LIN {X 0,Y 298.54,Z 403.296,A -85,B 0,C 180,E1 -16483.61,E2 -16483.61} C_VEL
LIN {X 0,Y 298.534,Z 403.297,A -85,B 0,C 180,E1 -16486.404,E2 -16486.404} C_VEL
LIN {X 0,Y 298.495,Z 403.302,A -85,B 0,C 180,E1 -16489.65,E2 -16489.65} C_VEL
LIN {X 0,Y 298.401,Z 403.314,A -85,B 0,C 180,E1 -16493.596,E2 -16493.596} C_VEL
LIN {X 0,Y 298.321,Z 403.323,A -85,B 0,C 180,E1 -16496.584,E2 -16496.584} C_VEL
LIN {X 0,Y 297.954,Z 403.371,A -85,B 0,C 180,E1 -16499.685,E2 -16499.685} C_VEL
LIN {X 0,Y 297.517,Z 403.428,A -85,B 0,C 180,E1 -16502.902,E2 -16502.902} C_VEL
LIN {X 0,Y 297.315,Z 403.659,A -85,B 0,C 180,E1 -16504.556,E2 -16504.556} C_VEL
LIN {X 0,Y 297.205,Z 406.502,A -85,B 0,C 180,E1 -16507.931,E2 -16507.931} C_VEL
LIN {X 0,Y 297.211,Z 408.026,A -85,B 0,C 180,E1 -16509.558,E2 -16509.558} C_VEL
LIN {X 0,Y 300.389,Z 421.173,A -85,B 0,C 180,E1 -16510.429,E2 -16510.429} C_VEL
LIN {X 0,Y 303.208,Z 434.297,A -85,B 0,C 180,E1 -16511.559,E2 -16511.559} C_VEL
LIN {X 0,Y 304.476,Z 441.111,A -85,B 0,C 180,E1 -16512.256,E2 -16512.256} C_VEL
LIN {X 0,Y 303.235,Z 453.565,A -85,B 0,C 180,E1 -16513.594,E2 -16513.594} C_VEL
LIN {X 0,Y 302.004,Z 464.15,A -85,B 0,C 180,E1 -16515.022,E2 -16515.022} C_VEL
LIN {X 0,Y 300.91,Z 473.555,A -85,B 0,C 180,E1 -16516.59,E2 -16516.59} C_VEL
LIN {X 0,Y 299.618,Z 483.514,A -85,B 0,C 180,E1 -16518.634,E2 -16518.634} C_VEL
LIN {X 0,Y 298.679,Z 491.025,A -85,B 0,C 180,E1 -16520.558,E2 -16520.558} C_VEL
LIN {X 0,Y 297.874,Z 498.058,A -85,B 0,C 180,E1 -16522.831,E2 -16522.831} C_VEL
LIN {X 0,Y 297.405,Z 502.476,A -85,B 0,C 180,E1 -16524.624,E2 -16524.624} C_VEL
LIN {X 0,Y 296.973,Z 507.02,A -85,B 0,C 180,E1 -16527.024,E2 -16527.024} C_VEL
LIN {X 0,Y 296.702,Z 509.213,A -85,B 0,C 180,E1 -16528.594,E2 -16528.594} C_VEL
LIN {X 0,Y 296.597,Z 511.611,A -85,B 0,C 180,E1 -16531.237,E2 -16531.237} C_VEL
LIN {X 0,Y 296.595,Z 512.398,A -85,B 0,C 180,E1 -16533.244,E2 -16533.244} C_VEL
LIN {X 0,Y 296.774,Z 512.436,A -85,B 0,C 180,E1 -16534.771,E2 -16534.771} C_VEL
LIN {X 0,Y 297.237,Z 511.374,A -85,B 0,C 180,E1 -16537.223,E2 -16537.223} C_VEL
LIN {X 0,Y 297.865,Z 509.479,A -85,B 0,C 180,E1 -16539.274,E2 -16539.274} C_VEL
LIN {X 0,Y 298.691,Z 506.354,A -85,B 0,C 180,E1 -16541.481,E2 -16541.481} C_VEL
LIN {X 0,Y 299.914,Z 501.581,A -85,B 0,C 180,E1 -16543.874,E2 -16543.874} C_VEL
LIN {X 0,Y 301.541,Z 495.408,A -85,B 0,C 180,E1 -16546.18,E2 -16546.18} C_VEL
LIN {X 0,Y 303.291,Z 488.055,A -85,B 0,C 180,E1 -16548.303,E2 -16548.303} C_VEL
LIN {X 0,Y 305.109,Z 480.486,A -85,B 0,C 180,E1 -16550.053,E2 -16550.053} C_VEL
LIN {X 0,Y 307.147,Z 471.173,A -85,B 0,C 180,E1 -16551.823,E2 -16551.823} C_VEL
LIN {X 0,Y 309.342,Z 460.153,A -85,B 0,C 180,E1 -16553.479,E2 -16553.479} C_VEL
LIN {X 0,Y 310.412,Z 454.213,A -85,B 0,C 180,E1 -16554.23,E2 -16554.23} C_VEL
LIN {X 0,Y 310.495,Z 451.09,A -85,B 0,C 180,E1 -16554.656,E2 -16554.656} C_VEL
LIN {X 0,Y 309.213,Z 446.849,A -85,B 0,C 180,E1 -16555.373,E2 -16555.373} C_VEL
LIN {X 0,Y 306.912,Z 443.084,A -85,B 0,C 180,E1 -16556.121,E2 -16556.121} C_VEL
LIN {X 0,Y 301.408,Z 435.464,A -85,B 0,C 180,E1 -16557.657,E2 -16557.657} C_VEL
LIN {X 0,Y 299.994,Z 432.52,A -85,B 0,C 180,E1 -16558.139,E2 -16558.139} C_VEL
LIN {X 0,Y 294.566,Z 419.508,A -85,B 0,C 180,E1 -16560.087,E2 -16560.087} C_VEL
LIN {X 0,Y 293.298,Z 416.848,A -85,B 0,C 180,E1 -16560.473,E2 -16560.473} C_VEL
LIN {X 0,Y 292.122,Z 413.899,A -85,B 0,C 180,E1 -16560.863,E2 -16560.863} C_VEL
LIN {X 0,Y 292.037,Z 413.448,A -85,B 0,C 180,E1 -16560.949,E2 -16560.949} C_VEL
LIN {X 0,Y 292.102,Z 411.884,A -85,B 0,C 180,E1 -16564.14,E2 -16564.14} C_VEL
LIN {X 0,Y 292.37,Z 410.624,A -85,B 0,C 180,E1 -16566.904,E2 -16566.904} C_VEL
LIN {X 0,Y 292.432,Z 409.493,A -85,B 0,C 180,E1 -16569.859,E2 -16569.859} C_VEL
LIN {X 0,Y 292.138,Z 408.34,A -85,B 0,C 180,E1 -16573.921,E2 -16573.921} C_VEL
LIN {X 0,Y 292.041,Z 407.747,A -85,B 0,C 180,E1 -16576.786,E2 -16576.786} C_VEL
LIN {X 0,Y 291.975,Z 407.316,A -85,B 0,C 180,E1 -16580.177,E2 -16580.177} C_VEL
LIN {X 0,Y 291.967,Z 407.269,A -85,B 0,C 180,E1 -16584.156,E2 -16584.156} C_VEL
LIN {X 0,Y 292.013,Z 407.587,A -85,B 0,C 180,E1 -16587.213,E2 -16587.213} C_VEL
LIN {X 0,Y 292.068,Z 408.231,A -85,B 0,C 180,E1 -16590.354,E2 -16590.354} C_VEL
LIN {X 0,Y 292.244,Z 409.294,A -85,B 0,C 180,E1 -16593.582,E2 -16593.582} C_VEL
LIN {X 0,Y 292.592,Z 411.114,A -85,B 0,C 180,E1 -16597.577,E2 -16597.577} C_VEL
LIN {X 0,Y 292.906,Z 412.784,A -85,B 0,C 180,E1 -16600.38,E2 -16600.38} C_VEL
LIN {X 0,Y 293.404,Z 415.441,A -85,B 0,C 180,E1 -16604.07,E2 -16604.07} C_VEL
LIN {X 0,Y 293.953,Z 418.857,A -85,B 0,C 180,E1 -16607.985,E2 -16607.985} C_VEL
LIN {X 0,Y 294.409,Z 422.603,A -85,B 0,C 180,E1 -16611.644,E2 -16611.644} C_VEL
LIN {X 0,Y 294.307,Z 425.693,A -85,B 0,C 180,E1 -16614.285,E2 -16614.285} C_VEL
LIN {X 0,Y 293.028,Z 430.824,A -85,B 0,C 180,E1 -16618.16,E2 -16618.16} C_VEL
LIN {X 0,Y 292.222,Z 434.847,A -85,B 0,C 180,E1 -16621.038,E2 -16621.038} C_VEL
LIN {X 0,Y 293.241,Z 438.506,A -85,B 0,C 180,E1 -16621.432,E2 -16621.432} C_VEL
LIN {X 0,Y 296.189,Z 447.824,A -85,B 0,C 180,E1 -16622.521,E2 -16622.521} C_VEL
LIN {X 0,Y 299.074,Z 460.374,A -85,B 0,C 180,E1 -16623.974,E2 -16623.974} C_VEL
LIN {X 0,Y 300.545,Z 472.286,A -85,B 0,C 180,E1 -16625.426,E2 -16625.426} C_VEL
LIN {X 0,Y 300.842,Z 482.738,A -85,B 0,C 180,E1 -16626.789,E2 -16626.789} C_VEL
LIN {X 0,Y 300.143,Z 492.535,A -85,B 0,C 180,E1 -16628.184,E2 -16628.184} C_VEL
LIN {X 0,Y 298.035,Z 501.95,A -85,B 0,C 180,E1 -16629.652,E2 -16629.652} C_VEL
LIN {X 0,Y 295.564,Z 512.297,A -85,B 0,C 180,E1 -16631.641,E2 -16631.641} C_VEL
LIN {X 0,Y 293.71,Z 520.668,A -85,B 0,C 180,E1 -16633.676,E2 -16633.676} C_VEL
LIN {X 0,Y 292.256,Z 527.544,A -85,B 0,C 180,E1 -16635.736,E2 -16635.736} C_VEL
LIN {X 0,Y 290.836,Z 533.963,A -85,B 0,C 180,E1 -16638.153,E2 -16638.153} C_VEL
LIN {X 0,Y 290.116,Z 538.211,A -85,B 0,C 180,E1 -16640.242,E2 -16640.242} C_VEL
LIN {X 0,Y 289.828,Z 540.46,A -85,B 0,C 180,E1 -16641.64,E2 -16641.64} C_VEL
LIN {X 0,Y 289.518,Z 543.698,A -85,B 0,C 180,E1 -16644.433,E2 -16644.433} C_VEL
LIN {X 0,Y 289.534,Z 544.718,A -85,B 0,C 180,E1 -16645.829,E2 -16645.829} C_VEL
LIN {X 0,Y 289.561,Z 545.291,A -85,B 0,C 180,E1 -16647.223,E2 -16647.223} C_VEL
LIN {X 0,Y 289.811,Z 545.227,A -85,B 0,C 180,E1 -16650.005,E2 -16650.005} C_VEL
LIN {X 0,Y 289.704,Z 544.575,A -85,B 0,C 180,E1 -16651.395,E2 -16651.395} C_VEL
LIN {X 0,Y 289.616,Z 543.459,A -85,B 0,C 180,E1 -16652.787,E2 -16652.787} C_VEL
LIN {X 0,Y 289.663,Z 541.916,A -85,B 0,C 180,E1 -16654.179,E2 -16654.179} C_VEL
LIN {X 0,Y 289.681,Z 539.425,A -85,B 0,C 180,E1 -16655.888,E2 -16655.888} C_VEL
LIN {X 0,Y 289.868,Z 534.452,A -85,B 0,C 180,E1 -16658.37,E2 -16658.37} C_VEL
LIN {X 0,Y 290.274,Z 528.94,A -85,B 0,C 180,E1 -16660.467,E2 -16660.467} C_VEL
LIN {X 0,Y 290.98,Z 522.039,A -85,B 0,C 180,E1 -16662.56,E2 -16662.56} C_VEL
LIN {X 0,Y 291.798,Z 514.992,A -85,B 0,C 180,E1 -16664.297,E2 -16664.297} C_VEL
LIN {X 0,Y 292.636,Z 506.875,A -85,B 0,C 180,E1 -16665.961,E2 -16665.961} C_VEL
LIN {X 0,Y 294.068,Z 497.254,A -85,B 0,C 180,E1 -16667.566,E2 -16667.566} C_VEL
LIN {X 0,Y 295.416,Z 485.913,A -85,B 0,C 180,E1 -16669.098,E2 -16669.098} C_VEL
LIN {X 0,Y 294.777,Z 474.417,A -85,B 0,C 180,E1 -16670.412,E2 -16670.412} C_VEL
LIN {X 0,Y 293.431,Z 461.228,A -85,B 0,C 180,E1 -16671.612,E2 -16671.612} C_VEL
LIN {X 0,Y 291.781,Z 447.799,A -85,B 0,C 180,E1 -16672.555,E2 -16672.555} C_VEL
LIN {X 0,Y 290.651,Z 439.673,A -85,B 0,C 180,E1 -16673.019,E2 -16673.019} C_VEL
LIN {X 0,Y 291.447,Z 432.932,A -85,B 0,C 180,E1 -16677.274,E2 -16677.274} C_VEL
LIN {X 0,Y 292.325,Z 426.915,A -85,B 0,C 180,E1 -16681.129,E2 -16681.129} C_VEL
LIN {X 0,Y 293.176,Z 422.072,A -85,B 0,C 180,E1 -16684.292,E2 -16684.292} C_VEL
LIN {X 0,Y 293.704,Z 418.403,A -85,B 0,C 180,E1 -16686.748,E2 -16686.748} C_VEL
LIN {X 0,Y 293.176,Z 413.948,A -85,B 0,C 180,E1 -16689.904,E2 -16689.904} C_VEL
LIN {X 0,Y 292.115,Z 408.18,A -85,B 0,C 180,E1 -16694.249,E2 -16694.249} C_VEL
LIN {X 0,Y 291.373,Z 404.192,A -85,B 0,C 180,E1 -16697.516,E2 -16697.516} C_VEL
LIN {X 0,Y 291.351,Z 404.195,A -85,B 0,C 180,E1 -16701.157,E2 -16701.157} C_VEL
LIN {X 0,Y 291.372,Z 404.188,A -85,B 0,C 180,E1 -16704.626,E2 -16704.626} C_VEL
LIN {X 0,Y 291.383,Z 404.186,A -85,B 0,C 180,E1 -16707.951,E2 -16707.951} C_VEL
LIN {X 0,Y 291.362,Z 404.193,A -85,B 0,C 180,E1 -16711.155,E2 -16711.155} C_VEL
LIN {X 0,Y 291.376,Z 404.186,A -85,B 0,C 180,E1 -16714.267,E2 -16714.267} C_VEL
LIN {X 0,Y 291.38,Z 404.19,A -85,B 0,C 180,E1 -16717.298,E2 -16717.298} C_VEL
LIN {X 0,Y 291.408,Z 404.183,A -85,B 0,C 180,E1 -16720.265,E2 -16720.265} C_VEL
LIN {X 0,Y 291.515,Z 404.172,A -85,B 0,C 180,E1 -16724.665,E2 -16724.665} C_VEL
LIN {X 0,Y 291.545,Z 404.17,A -85,B 0,C 180,E1 -16728.88,E2 -16728.88} C_VEL
LIN {X 0,Y 291.682,Z 404.149,A -85,B 0,C 180,E1 -16731.687,E2 -16731.687} C_VEL
LIN {X 0,Y 291.627,Z 404.157,A -85,B 0,C 180,E1 -16734.467,E2 -16734.467} C_VEL
LIN {X 0,Y 291.9,Z 404.124,A -85,B 0,C 180,E1 -16738.619,E2 -16738.619} C_VEL
LIN {X 0,Y 291.896,Z 404.124,A -85,B 0,C 180,E1 -16741.378,E2 -16741.378} C_VEL
LIN {X 0,Y 291.701,Z 404.151,A -85,B 0,C 180,E1 -16746.918,E2 -16746.918} C_VEL
LIN {X 0,Y 291.582,Z 404.161,A -85,B 0,C 180,E1 -16749.712,E2 -16749.712} C_VEL
LIN {X 0,Y 291.528,Z 404.168,A -85,B 0,C 180,E1 -16753.949,E2 -16753.949} C_VEL
LIN {X 0,Y 291.441,Z 404.184,A -85,B 0,C 180,E1 -16756.819,E2 -16756.819} C_VEL
LIN {X 0,Y 291.405,Z 404.184,A -85,B 0,C 180,E1 -16759.84,E2 -16759.84} C_VEL
LIN {X 0,Y 291.394,Z 404.185,A -85,B 0,C 180,E1 -16764.204,E2 -16764.204} C_VEL
LIN {X 0,Y 291.424,Z 404.182,A -85,B 0,C 180,E1 -16767.27,E2 -16767.27} C_VEL
LIN {X 0,Y 291.334,Z 404.195,A -85,B 0,C 180,E1 -16770.436,E2 -16770.436} C_VEL
LIN {X 0,Y 291.354,Z 404.189,A -85,B 0,C 180,E1 -16773.695,E2 -16773.695} C_VEL
LIN {X 0,Y 291.378,Z 404.187,A -85,B 0,C 180,E1 -16777.249,E2 -16777.249} C_VEL
LIN {X 0,Y 291.34,Z 404.196,A -85,B 0,C 180,E1 -16780.639,E2 -16780.639} C_VEL
LIN {X 0,Y 291.299,Z 404.201,A -85,B 0,C 180,E1 -16784.398,E2 -16784.398} C_VEL
LIN {X 0,Y 291.324,Z 404.197,A -85,B 0,C 180,E1 -16788.403,E2 -16788.403} C_VEL
LIN {X 0,Y 291.353,Z 404.19,A -85,B 0,C 180,E1 -16791.153,E2 -16791.153} C_VEL
LIN {X 0,Y 291.366,Z 404.192,A -85,B 0,C 180,E1 -16794.622,E2 -16794.622} C_VEL
LIN {X 0,Y 291.375,Z 404.188,A -85,B 0,C 180,E1 -16797.946,E2 -16797.946} C_VEL
LIN {X 0,Y 291.381,Z 404.187,A -85,B 0,C 180,E1 -16801.153,E2 -16801.153} C_VEL
LIN {X 0,Y 291.417,Z 404.186,A -85,B 0,C 180,E1 -16804.267,E2 -16804.267} C_VEL
LIN {X 0,Y 291.39,Z 404.185,A -85,B 0,C 180,E1 -16807.296,E2 -16807.296} C_VEL
LIN {X 0,Y 291.459,Z 404.182,A -85,B 0,C 180,E1 -16810.266,E2 -16810.266} C_VEL
LIN {X 0,Y 291.555,Z 404.167,A -85,B 0,C 180,E1 -16814.619,E2 -16814.619} C_VEL
LIN {X 0,Y 291.533,Z 404.168,A -85,B 0,C 180,E1 -16818.876,E2 -16818.876} C_VEL
LIN {X 0,Y 291.684,Z 404.149,A -85,B 0,C 180,E1 -16821.683,E2 -16821.683} C_VEL
LIN {X 0,Y 291.621,Z 404.16,A -85,B 0,C 180,E1 -16824.463,E2 -16824.463} C_VEL
LIN {X 0,Y 291.882,Z 404.125,A -85,B 0,C 180,E1 -16828.615,E2 -16828.615} C_VEL
LIN {X 0,Y 291.882,Z 404.124,A -85,B 0,C 180,E1 -16831.375,E2 -16831.375} C_VEL
LIN {X 0,Y 291.736,Z 404.142,A -85,B 0,C 180,E1 -16836.913,E2 -16836.913} C_VEL
LIN {X 0,Y 291.618,Z 404.158,A -85,B 0,C 180,E1 -16839.707,E2 -16839.707} C_VEL
LIN {X 0,Y 291.509,Z 404.175,A -85,B 0,C 180,E1 -16843.945,E2 -16843.945} C_VEL
LIN {X 0,Y 291.472,Z 404.174,A -85,B 0,C 180,E1 -16846.813,E2 -16846.813} C_VEL
LIN {X 0,Y 291.434,Z 404.184,A -85,B 0,C 180,E1 -16849.87,E2 -16849.87} C_VEL
LIN {X 0,Y 291.331,Z 404.196,A -85,B 0,C 180,E1 -16854.205,E2 -16854.205} C_VEL
LIN {X 0,Y 291.17,Z 404.213,A -85,B 0,C 180,E1 -16857.29,E2 -16857.29} C_VEL
LIN {X 0,Y 290.798,Z 404.26,A -85,B 0,C 180,E1 -16860.492,E2 -16860.492} C_VEL
LIN {X 0,Y 290.267,Z 404.462,A -85,B 0,C 180,E1 -16864.595,E2 -16864.595} C_VEL
LIN {X 0,Y 290.182,Z 406.676,A -85,B 0,C 180,E1 -16867.256,E2 -16867.256} C_VEL
LIN {X 0,Y 290.127,Z 408.296,A -85,B 0,C 180,E1 -16869.152,E2 -16869.152} C_VEL
LIN {X 0,Y 293.307,Z 421.562,A -85,B 0,C 180,E1 -16870.063,E2 -16870.063} C_VEL
LIN {X 0,Y 296.094,Z 434.385,A -85,B 0,C 180,E1 -16871.19,E2 -16871.19} C_VEL
LIN {X 0,Y 297.463,Z 441.449,A -85,B 0,C 180,E1 -16871.927,E2 -16871.927} C_VEL
LIN {X 0,Y 296.397,Z 453.238,A -85,B 0,C 180,E1 -16873.223,E2 -16873.223} C_VEL
LIN {X 0,Y 295.019,Z 464.665,A -85,B 0,C 180,E1 -16874.792,E2 -16874.792} C_VEL
LIN {X 0,Y 293.793,Z 474.842,A -85,B 0,C 180,E1 -16876.55,E2 -16876.55} C_VEL
LIN {X 0,Y 292.664,Z 483.398,A -85,B 0,C 180,E1 -16878.357,E2 -16878.357} C_VEL
LIN {X 0,Y 291.632,Z 491.429,A -85,B 0,C 180,E1 -16880.448,E2 -16880.448} C_VEL
LIN {X 0,Y 290.783,Z 498.61,A -85,B 0,C 180,E1 -16882.828,E2 -16882.828} C_VEL
LIN {X 0,Y 290.182,Z 504.563,A -85,B 0,C 180,E1 -16885.42,E2 -16885.42} C_VEL
LIN {X 0,Y 289.766,Z 508.44,A -85,B 0,C 180,E1 -16887.753,E2 -16887.753} C_VEL
LIN {X 0,Y 289.531,Z 510.403,A -85,B 0,C 180,E1 -16889.355,E2 -16889.355} C_VEL
LIN {X 0,Y 289.51,Z 511.762,A -85,B 0,C 180,E1 -16890.956,E2 -16890.956} C_VEL
LIN {X 0,Y 289.484,Z 512.601,A -85,B 0,C 180,E1 -16892.532,E2 -16892.532} C_VEL
LIN {X 0,Y 289.593,Z 512.914,A -85,B 0,C 180,E1 -16894.1,E2 -16894.1} C_VEL
LIN {X 0,Y 289.827,Z 512.705,A -85,B 0,C 180,E1 -16895.656,E2 -16895.656} C_VEL
LIN {X 0,Y 290.148,Z 512.042,A -85,B 0,C 180,E1 -16897.199,E2 -16897.199} C_VEL
LIN {X 0,Y 290.601,Z 510.841,A -85,B 0,C 180,E1 -16898.731,E2 -16898.731} C_VEL
LIN {X 0,Y 291.445,Z 508.149,A -85,B 0,C 180,E1 -16901.012,E2 -16901.012} C_VEL
LIN {X 0,Y 292.503,Z 504.355,A -85,B 0,C 180,E1 -16903.244,E2 -16903.244} C_VEL
LIN {X 0,Y 293.941,Z 499.288,A -85,B 0,C 180,E1 -16905.462,E2 -16905.462} C_VEL
LIN {X 0,Y 295.677,Z 492.842,A -85,B 0,C 180,E1 -16907.649,E2 -16907.649} C_VEL
LIN {X 0,Y 297.735,Z 484.762,A -85,B 0,C 180,E1 -16909.804,E2 -16909.804} C_VEL
LIN {X 0,Y 299.825,Z 476.1,A -85,B 0,C 180,E1 -16911.654,E2 -16911.654} C_VEL
LIN {X 0,Y 302.063,Z 466.318,A -85,B 0,C 180,E1 -16913.321,E2 -16913.321} C_VEL
LIN {X 0,Y 304.207,Z 455.212,A -85,B 0,C 180,E1 -16914.845,E2 -16914.845} C_VEL
LIN {X 0,Y 304.748,Z 451.943,A -85,B 0,C 180,E1 -16915.234,E2 -16915.234} C_VEL
LIN {X 0,Y 303.135,Z 442.861,A -85,B 0,C 180,E1 -16916.605,E2 -16916.605} C_VEL
LIN {X 0,Y 300.794,Z 434.624,A -85,B 0,C 180,E1 -16917.825,E2 -16917.825} C_VEL
LIN {X 0,Y 299.994,Z 432.52,A -85,B 0,C 180,E1 -16918.139,E2 -16918.139} C_VEL
LIN {X 0,Y 298.406,Z 429.93,A -85,B 0,C 180,E1 -16918.623,E2 -16918.623} C_VEL
LIN {X 0,Y 294.556,Z 426.882,A -85,B 0,C 180,E1 -16919.5,E2 -16919.5} C_VEL
LIN {X 0,Y 289.838,Z 423.293,A -85,B 0,C 180,E1 -16920.59,E2 -16920.59} C_VEL
LIN {X 0,Y 288.637,Z 421.64,A -85,B 0,C 180,E1 -16920.936,E2 -16920.936} C_VEL
LIN {X 0,Y 286.733,Z 417.71,A -85,B 0,C 180,E1 -16921.581,E2 -16921.581} C_VEL
LIN {X 0,Y 285.365,Z 415.042,A -85,B 0,C 180,E1 -16922.03,E2 -16922.03} C_VEL
LIN {X 0,Y 285.135,Z 414.1,A -85,B 0,C 180,E1 -16922.164,E2 -16922.164} C_VEL
LIN {X 0,Y 285.417,Z 411.93,A -85,B 0,C 180,E1 -16927.073,E2 -16927.073} C_VEL
LIN {X 0,Y 285.465,Z 410.859,A -85,B 0,C 180,E1 -16930.049,E2 -16930.049} C_VEL
LIN {X 0,Y 285.193,Z 409.742,A -85,B 0,C 180,E1 -16934.268,E2 -16934.268} C_VEL
LIN {X 0,Y 285.083,Z 409.215,A -85,B 0,C 180,E1 -16937.209,E2 -16937.209} C_VEL
LIN {X 0,Y 285.029,Z 408.873,A -85,B 0,C 180,E1 -16940.471,E2 -16940.471} C_VEL
LIN {X 0,Y 285.044,Z 408.927,A -85,B 0,C 180,E1 -16944.782,E2 -16944.782} C_VEL
LIN {X 0,Y 285.095,Z 409.333,A -85,B 0,C 180,E1 -16947.93,E2 -16947.93} C_VEL
LIN {X 0,Y 285.185,Z 410.122,A -85,B 0,C 180,E1 -16951.167,E2 -16951.167} C_VEL
LIN {X 0,Y 285.395,Z 411.308,A -85,B 0,C 180,E1 -16954.5,E2 -16954.5} C_VEL
LIN {X 0,Y 285.722,Z 413.027,A -85,B 0,C 180,E1 -16958.094,E2 -16958.094} C_VEL
LIN {X 0,Y 286.142,Z 415.15,A -85,B 0,C 180,E1 -16961.542,E2 -16961.542} C_VEL
LIN {X 0,Y 286.61,Z 417.989,A -85,B 0,C 180,E1 -16965.327,E2 -16965.327} C_VEL
LIN {X 0,Y 287.177,Z 421.618,A -85,B 0,C 180,E1 -16969.347,E2 -16969.347} C_VEL
LIN {X 0,Y 287.473,Z 424.723,A -85,B 0,C 180,E1 -16972.332,E2 -16972.332} C_VEL
LIN {X 0,Y 287.336,Z 426.692,A -85,B 0,C 180,E1 -16974.062,E2 -16974.062} C_VEL
LIN {X 0,Y 285.995,Z 431.899,A -85,B 0,C 180,E1 -16978.114,E2 -16978.114} C_VEL
LIN {X 0,Y 285.481,Z 434.281,A -85,B 0,C 180,E1 -16979.875,E2 -16979.875} C_VEL
LIN {X 0,Y 286.353,Z 437.614,A -85,B 0,C 180,E1 -16980.236,E2 -16980.236} C_VEL
LIN {X 0,Y 287.246,Z 440.024,A -85,B 0,C 180,E1 -16980.56,E2 -16980.56} C_VEL
LIN {X 0,Y 289.964,Z 448.634,A -85,B 0,C 180,E1 -16981.628,E2 -16981.628} C_VEL
LIN {X 0,Y 292.563,Z 459.973,A -85,B 0,C 180,E1 -16983.052,E2 -16983.052} C_VEL
LIN {X 0,Y 294.099,Z 471.5,A -85,B 0,C 180,E1 -16984.53,E2 -16984.53} C_VEL
LIN {X 0,Y 294.512,Z 481.31,A -85,B 0,C 180,E1 -16985.867,E2 -16985.867} C_VEL
LIN {X 0,Y 293.826,Z 492.303,A -85,B 0,C 180,E1 -16987.505,E2 -16987.505} C_VEL
LIN {X 0,Y 291.436,Z 502.634,A -85,B 0,C 180,E1 -16989.17,E2 -16989.17} C_VEL
LIN {X 0,Y 289.285,Z 511.205,A -85,B 0,C 180,E1 -16990.86,E2 -16990.86} C_VEL
LIN {X 0,Y 287.151,Z 519.685,A -85,B 0,C 180,E1 -16992.926,E2 -16992.926} C_VEL
LIN {X 0,Y 285.645,Z 526.607,A -85,B 0,C 180,E1 -16995.034,E2 -16995.034} C_VEL
LIN {X 0,Y 284.17,Z 532.269,A -85,B 0,C 180,E1 -16997.145,E2 -16997.145} C_VEL
LIN {X 0,Y 283.318,Z 536.789,A -85,B 0,C 180,E1 -16999.284,E2 -16999.284} C_VEL
LIN {X 0,Y 282.774,Z 540.265,A -85,B 0,C 180,E1 -17001.429,E2 -17001.429} C_VEL
LIN {X 0,Y 282.441,Z 543.413,A -85,B 0,C 180,E1 -17004.293,E2 -17004.293} C_VEL
LIN {X 0,Y 282.432,Z 544.36,A -85,B 0,C 180,E1 -17005.724,E2 -17005.724} C_VEL
LIN {X 0,Y 282.484,Z 544.887,A -85,B 0,C 180,E1 -17007.153,E2 -17007.153} C_VEL
LIN {X 0,Y 282.723,Z 544.75,A -85,B 0,C 180,E1 -17010.005,E2 -17010.005} C_VEL
LIN {X 0,Y 282.615,Z 544.032,A -85,B 0,C 180,E1 -17011.43,E2 -17011.43} C_VEL
LIN {X 0,Y 282.542,Z 542.863,A -85,B 0,C 180,E1 -17012.857,E2 -17012.857} C_VEL
LIN {X 0,Y 282.553,Z 539.929,A -85,B 0,C 180,E1 -17015.256,E2 -17015.256} C_VEL
LIN {X 0,Y 282.725,Z 535.248,A -85,B 0,C 180,E1 -17017.863,E2 -17017.863} C_VEL
LIN {X 0,Y 283.174,Z 529.036,A -85,B 0,C 180,E1 -17020.371,E2 -17020.371} C_VEL
LIN {X 0,Y 283.838,Z 522.241,A -85,B 0,C 180,E1 -17022.518,E2 -17022.518} C_VEL
LIN {X 0,Y 284.672,Z 515.319,A -85,B 0,C 180,E1 -17024.298,E2 -17024.298} C_VEL
LIN {X 0,Y 285.459,Z 508.77,A -85,B 0,C 180,E1 -17025.718,E2 -17025.718} C_VEL
LIN {X 0,Y 286.65,Z 500.109,A -85,B 0,C 180,E1 -17027.299,E2 -17027.299} C_VEL
LIN {X 0,Y 288.003,Z 489.614,A -85,B 0,C 180,E1 -17028.869,E2 -17028.869} C_VEL
LIN {X 0,Y 288.427,Z 484.086,A -85,B 0,C 180,E1 -17029.58,E2 -17029.58} C_VEL
LIN {X 0,Y 287.45,Z 471.326,A -85,B 0,C 180,E1 -17031.016,E2 -17031.016} C_VEL
LIN {X 0,Y 286.077,Z 458.16,A -85,B 0,C 180,E1 -17032.197,E2 -17032.197} C_VEL
LIN {X 0,Y 284.204,Z 443.767,A -85,B 0,C 180,E1 -17033.163,E2 -17033.163} C_VEL
LIN {X 0,Y 283.628,Z 439.323,A -85,B 0,C 180,E1 -17033.421,E2 -17033.421} C_VEL
LIN {X 0,Y 284.512,Z 432.291,A -85,B 0,C 180,E1 -17037.996,E2 -17037.996} C_VEL
LIN {X 0,Y 285.724,Z 425.101,A -85,B 0,C 180,E1 -17042.766,E2 -17042.766} C_VEL
LIN {X 0,Y 286.525,Z 420.229,A -85,B 0,C 180,E1 -17046.068,E2 -17046.068} C_VEL
LIN {X 0,Y 286.477,Z 417.12,A -85,B 0,C 180,E1 -17048.274,E2 -17048.274} C_VEL
LIN {X 0,Y 285.733,Z 412.65,A -85,B 0,C 180,E1 -17051.619,E2 -17051.619} C_VEL
LIN {X 0,Y 284.775,Z 407.454,A -85,B 0,C 180,E1 -17055.706,E2 -17055.706} C_VEL
LIN {X 0,Y 284.329,Z 405.07,A -85,B 0,C 180,E1 -17057.774,E2 -17057.774} C_VEL
LIN {X 0,Y 284.325,Z 405.065,A -85,B 0,C 180,E1 -17062.284,E2 -17062.284} C_VEL
LIN {X 0,Y 284.324,Z 405.068,A -85,B 0,C 180,E1 -17065.352,E2 -17065.352} C_VEL
LIN {X 0,Y 284.302,Z 405.07,A -85,B 0,C 180,E1 -17068.725,E2 -17068.725} C_VEL
LIN {X 0,Y 284.301,Z 405.068,A -85,B 0,C 180,E1 -17071.985,E2 -17071.985} C_VEL
LIN {X 0,Y 284.339,Z 405.064,A -85,B 0,C 180,E1 -17076.148,E2 -17076.148} C_VEL
LIN {X 0,Y 284.352,Z 405.062,A -85,B 0,C 180,E1 -17079.928,E2 -17079.928} C_VEL
LIN {X 0,Y 284.464,Z 405.049,A -85,B 0,C 180,E1 -17084.493,E2 -17084.493} C_VEL
LIN {X 0,Y 284.482,Z 405.048,A -85,B 0,C 180,E1 -17088.6,E2 -17088.6} C_VEL
LIN {X 0,Y 284.637,Z 405.027,A -85,B 0,C 180,E1 -17091.479,E2 -17091.479} C_VEL
LIN {X 0,Y 284.597,Z 405.032,A -85,B 0,C 180,E1 -17094.33,E2 -17094.33} C_VEL
LIN {X 0,Y 284.866,Z 404.999,A -85,B 0,C 180,E1 -17098.585,E2 -17098.585} C_VEL
LIN {X 0,Y 284.862,Z 405,A -85,B 0,C 180,E1 -17101.412,E2 -17101.412} C_VEL
LIN {X 0,Y 284.656,Z 405.026,A -85,B 0,C 180,E1 -17107.09,E2 -17107.09} C_VEL
LIN {X 0,Y 284.529,Z 405.04,A -85,B 0,C 180,E1 -17109.955,E2 -17109.955} C_VEL
LIN {X 0,Y 284.477,Z 405.047,A -85,B 0,C 180,E1 -17114.302,E2 -17114.302} C_VEL
LIN {X 0,Y 284.346,Z 405.068,A -85,B 0,C 180,E1 -17118.741,E2 -17118.741} C_VEL
LIN {X 0,Y 284.345,Z 405.063,A -85,B 0,C 180,E1 -17123.293,E2 -17123.293} C_VEL
LIN {X 0,Y 284.402,Z 405.057,A -85,B 0,C 180,E1 -17127.168,E2 -17127.168} C_VEL
LIN {X 0,Y 284.298,Z 405.068,A -85,B 0,C 180,E1 -17131.272,E2 -17131.272} C_VEL
LIN {X 0,Y 284.351,Z 405.063,A -85,B 0,C 180,E1 -17135.344,E2 -17135.344} C_VEL
LIN {X 0,Y 284.315,Z 405.068,A -85,B 0,C 180,E1 -17138.167,E2 -17138.167} C_VEL
LIN {X 0,Y 284.277,Z 405.073,A -85,B 0,C 180,E1 -17142.12,E2 -17142.12} C_VEL
LIN {X 0,Y 284.263,Z 405.075,A -85,B 0,C 180,E1 -17146.185,E2 -17146.185} C_VEL
LIN {X 0,Y 284.313,Z 405.068,A -85,B 0,C 180,E1 -17150.02,E2 -17150.02} C_VEL
LIN {X 0,Y 284.336,Z 405.064,A -85,B 0,C 180,E1 -17153.61,E2 -17153.61} C_VEL
LIN {X 0,Y 284.312,Z 405.066,A -85,B 0,C 180,E1 -17157.185,E2 -17157.185} C_VEL
LIN {X 0,Y 284.359,Z 405.066,A -85,B 0,C 180,E1 -17160.371,E2 -17160.371} C_VEL
LIN {X 0,Y 284.379,Z 405.059,A -85,B 0,C 180,E1 -17163.582,E2 -17163.582} C_VEL
LIN {X 0,Y 284.371,Z 405.062,A -85,B 0,C 180,E1 -17166.703,E2 -17166.703} C_VEL
LIN {X 0,Y 284.403,Z 405.055,A -85,B 0,C 180,E1 -17171.257,E2 -17171.257} C_VEL
LIN {X 0,Y 284.492,Z 405.048,A -85,B 0,C 180,E1 -17174.454,E2 -17174.454} C_VEL
LIN {X 0,Y 284.485,Z 405.048,A -85,B 0,C 180,E1 -17178.596,E2 -17178.596} C_VEL
LIN {X 0,Y 284.635,Z 405.026,A -85,B 0,C 180,E1 -17181.475,E2 -17181.475} C_VEL
LIN {X 0,Y 284.592,Z 405.036,A -85,B 0,C 180,E1 -17184.326,E2 -17184.326} C_VEL
LIN {X 0,Y 284.848,Z 405.002,A -85,B 0,C 180,E1 -17188.581,E2 -17188.581} C_VEL
LIN {X 0,Y 284.848,Z 405,A -85,B 0,C 180,E1 -17191.409,E2 -17191.409} C_VEL
LIN {X 0,Y 284.688,Z 405.02,A -85,B 0,C 180,E1 -17197.085,E2 -17197.085} C_VEL
LIN {X 0,Y 284.555,Z 405.04,A -85,B 0,C 180,E1 -17199.95,E2 -17199.95} C_VEL
LIN {X 0,Y 284.469,Z 405.05,A -85,B 0,C 180,E1 -17204.298,E2 -17204.298} C_VEL
LIN {X 0,Y 284.41,Z 405.054,A -85,B 0,C 180,E1 -17207.243,E2 -17207.243} C_VEL
LIN {X 0,Y 284.362,Z 405.064,A -85,B 0,C 180,E1 -17210.237,E2 -17210.237} C_VEL
LIN {X 0,Y 284.298,Z 405.073,A -85,B 0,C 180,E1 -17213.846,E2 -17213.846} C_VEL
LIN {X 0,Y 284.156,Z 405.087,A -85,B 0,C 180,E1 -17217.082,E2 -17217.082} C_VEL
LIN {X 0,Y 283.818,Z 405.134,A -85,B 0,C 180,E1 -17219.928,E2 -17219.928} C_VEL
LIN {X 0,Y 283.375,Z 405.19,A -85,B 0,C 180,E1 -17223.06,E2 -17223.06} C_VEL
LIN {X 0,Y 283.198,Z 405.595,A -85,B 0,C 180,E1 -17225.023,E2 -17225.023} C_VEL
LIN {X 0,Y 283.068,Z 408.667,A -85,B 0,C 180,E1 -17228.729,E2 -17228.729} C_VEL
LIN {X 0,Y 286.585,Z 423.421,A -85,B 0,C 180,E1 -17229.8,E2 -17229.8} C_VEL
LIN {X 0,Y 289.315,Z 436.129,A -85,B 0,C 180,E1 -17230.978,E2 -17230.978} C_VEL
LIN {X 0,Y 290.535,Z 442.615,A -85,B 0,C 180,E1 -17231.69,E2 -17231.69} C_VEL
LIN {X 0,Y 289.41,Z 454.12,A -85,B 0,C 180,E1 -17232.996,E2 -17232.996} C_VEL
LIN {X 0,Y 288.109,Z 464.681,A -85,B 0,C 180,E1 -17234.481,E2 -17234.481} C_VEL
LIN {X 0,Y 286.739,Z 475.661,A -85,B 0,C 180,E1 -17236.424,E2 -17236.424} C_VEL
LIN {X 0,Y 285.53,Z 484.489,A -85,B 0,C 180,E1 -17238.352,E2 -17238.352} C_VEL
LIN {X 0,Y 284.516,Z 492.38,A -85,B 0,C 180,E1 -17240.503,E2 -17240.503} C_VEL
LIN {X 0,Y 283.665,Z 499.478,A -85,B 0,C 180,E1 -17242.944,E2 -17242.944} C_VEL
LIN {X 0,Y 283.12,Z 504.531,A -85,B 0,C 180,E1 -17245.186,E2 -17245.186} C_VEL
LIN {X 0,Y 282.678,Z 508.7,A -85,B 0,C 180,E1 -17247.693,E2 -17247.693} C_VEL
LIN {X 0,Y 282.422,Z 511.809,A -85,B 0,C 180,E1 -17250.557,E2 -17250.557} C_VEL
LIN {X 0,Y 282.382,Z 512.627,A -85,B 0,C 180,E1 -17251.78,E2 -17251.78} C_VEL
LIN {X 0,Y 282.458,Z 513.258,A -85,B 0,C 180,E1 -17253.588,E2 -17253.588} C_VEL
LIN {X 0,Y 282.618,Z 513.332,A -85,B 0,C 180,E1 -17254.993,E2 -17254.993} C_VEL
LIN {X 0,Y 282.966,Z 512.859,A -85,B 0,C 180,E1 -17256.758,E2 -17256.758} C_VEL
LIN {X 0,Y 283.327,Z 512.045,A -85,B 0,C 180,E1 -17258.158,E2 -17258.158} C_VEL
LIN {X 0,Y 284.013,Z 510.286,A -85,B 0,C 180,E1 -17260.085,E2 -17260.085} C_VEL
LIN {X 0,Y 285.17,Z 506.472,A -85,B 0,C 180,E1 -17262.8,E2 -17262.8} C_VEL
LIN {X 0,Y 286.564,Z 501.954,A -85,B 0,C 180,E1 -17265.079,E2 -17265.079} C_VEL
LIN {X 0,Y 288.343,Z 496.078,A -85,B 0,C 180,E1 -17267.33,E2 -17267.33} C_VEL
LIN {X 0,Y 290.392,Z 488.697,A -85,B 0,C 180,E1 -17269.543,E2 -17269.543} C_VEL
LIN {X 0,Y 292.628,Z 480.477,A -85,B 0,C 180,E1 -17271.501,E2 -17271.501} C_VEL
LIN {X 0,Y 294.691,Z 471.992,A -85,B 0,C 180,E1 -17273.153,E2 -17273.153} C_VEL
LIN {X 0,Y 297.217,Z 460.681,A -85,B 0,C 180,E1 -17274.914,E2 -17274.914} C_VEL
LIN {X 0,Y 298.554,Z 453.892,A -85,B 0,C 180,E1 -17275.797,E2 -17275.797} C_VEL
LIN {X 0,Y 296.915,Z 444.526,A -85,B 0,C 180,E1 -17277.288,E2 -17277.288} C_VEL
LIN {X 0,Y 294.422,Z 436.116,A -85,B 0,C 180,E1 -17278.633,E2 -17278.633} C_VEL
LIN {X 0,Y 289.273,Z 423.137,A -85,B 0,C 180,E1 -17280.698,E2 -17280.698} C_VEL
LIN {X 0,Y 288.637,Z 421.64,A -85,B 0,C 180,E1 -17280.936,E2 -17280.936} C_VEL
LIN {X 0,Y 286.721,Z 419.182,A -85,B 0,C 180,E1 -17281.48,E2 -17281.48} C_VEL
LIN {X 0,Y 282.593,Z 416.453,A -85,B 0,C 180,E1 -17282.465,E2 -17282.465} C_VEL
LIN {X 0,Y 279.586,Z 415.162,A -85,B 0,C 180,E1 -17283.355,E2 -17283.355} C_VEL
LIN {X 0,Y 278.296,Z 414.559,A -85,B 0,C 180,E1 -17284.122,E2 -17284.122} C_VEL
LIN {X 0,Y 278.199,Z 414.424,A -85,B 0,C 180,E1 -17284.393,E2 -17284.393} C_VEL
LIN {X 0,Y 278.478,Z 413.252,A -85,B 0,C 180,E1 -17287.25,E2 -17287.25} C_VEL
LIN {X 0,Y 278.502,Z 412.236,A -85,B 0,C 180,E1 -17290.25,E2 -17290.25} C_VEL
LIN {X 0,Y 278.258,Z 411.158,A -85,B 0,C 180,E1 -17294.631,E2 -17294.631} C_VEL
LIN {X 0,Y 278.149,Z 410.691,A -85,B 0,C 180,E1 -17297.651,E2 -17297.651} C_VEL
LIN {X 0,Y 278.092,Z 410.463,A -85,B 0,C 180,E1 -17300.78,E2 -17300.78} C_VEL
LIN {X 0,Y 278.137,Z 410.54,A -85,B 0,C 180,E1 -17304.559,E2 -17304.559} C_VEL
LIN {X 0,Y 278.192,Z 411.146,A -85,B 0,C 180,E1 -17308.687,E2 -17308.687} C_VEL
LIN {X 0,Y 278.328,Z 412.041,A -85,B 0,C 180,E1 -17312.025,E2 -17312.025} C_VEL
LIN {X 0,Y 278.61,Z 413.706,A -85,B 0,C 180,E1 -17316.187,E2 -17316.187} C_VEL
LIN {X 0,Y 278.905,Z 415.202,A -85,B 0,C 180,E1 -17319.049,E2 -17319.049} C_VEL
LIN {X 0,Y 279.378,Z 417.581,A -85,B 0,C 180,E1 -17322.783,E2 -17322.783} C_VEL
LIN {X 0,Y 279.877,Z 420.686,A -85,B 0,C 180,E1 -17326.739,E2 -17326.739} C_VEL
LIN {X 0,Y 280.235,Z 423.006,A -85,B 0,C 180,E1 -17329.312,E2 -17329.312} C_VEL
LIN {X 0,Y 280.45,Z 424.881,A -85,B 0,C 180,E1 -17331.216,E2 -17331.216} C_VEL
LIN {X 0,Y 280.406,Z 427.16,A -85,B 0,C 180,E1 -17333.327,E2 -17333.327} C_VEL
LIN {X 0,Y 279.66,Z 430.405,A -85,B 0,C 180,E1 -17336.029,E2 -17336.029} C_VEL
LIN {X 0,Y 278.838,Z 433.745,A -85,B 0,C 180,E1 -17338.6,E2 -17338.6} C_VEL
LIN {X 0,Y 279.777,Z 437.165,A -85,B 0,C 180,E1 -17338.997,E2 -17338.997} C_VEL
LIN {X 0,Y 280.747,Z 439.744,A -85,B 0,C 180,E1 -17339.366,E2 -17339.366} C_VEL
LIN {X 0,Y 283.699,Z 449.071,A -85,B 0,C 180,E1 -17340.647,E2 -17340.647} C_VEL
LIN {X 0,Y 286.378,Z 460.728,A -85,B 0,C 180,E1 -17342.214,E2 -17342.214} C_VEL
LIN {X 0,Y 287.834,Z 472.059,A -85,B 0,C 180,E1 -17343.771,E2 -17343.771} C_VEL
LIN {X 0,Y 288.164,Z 482.683,A -85,B 0,C 180,E1 -17345.3,E2 -17345.3} C_VEL
LIN {X 0,Y 287.353,Z 493.379,A -85,B 0,C 180,E1 -17346.969,E2 -17346.969} C_VEL
LIN {X 0,Y 284.86,Z 503.368,A -85,B 0,C 180,E1 -17348.666,E2 -17348.666} C_VEL
LIN {X 0,Y 282.167,Z 513.16,A -85,B 0,C 180,E1 -17350.736,E2 -17350.736} C_VEL
LIN {X 0,Y 280.059,Z 521.223,A -85,B 0,C 180,E1 -17352.857,E2 -17352.857} C_VEL
LIN {X 0,Y 278.794,Z 526.772,A -85,B 0,C 180,E1 -17354.657,E2 -17354.657} C_VEL
LIN {X 0,Y 277.239,Z 532.298,A -85,B 0,C 180,E1 -17356.818,E2 -17356.818} C_VEL
LIN {X 0,Y 276.301,Z 536.691,A -85,B 0,C 180,E1 -17359.008,E2 -17359.008} C_VEL
LIN {X 0,Y 275.712,Z 540.074,A -85,B 0,C 180,E1 -17361.208,E2 -17361.208} C_VEL
LIN {X 0,Y 275.484,Z 541.806,A -85,B 0,C 180,E1 -17362.677,E2 -17362.677} C_VEL
LIN {X 0,Y 275.344,Z 543.379,A -85,B 0,C 180,E1 -17364.544,E2 -17364.544} C_VEL
LIN {X 0,Y 275.408,Z 544.483,A -85,B 0,C 180,E1 -17367.08,E2 -17367.08} C_VEL
LIN {X 0,Y 275.458,Z 544.57,A -85,B 0,C 180,E1 -17368.543,E2 -17368.543} C_VEL
LIN {X 0,Y 275.637,Z 544.259,A -85,B 0,C 180,E1 -17370.005,E2 -17370.005} C_VEL
LIN {X 0,Y 275.527,Z 543.471,A -85,B 0,C 180,E1 -17371.467,E2 -17371.467} C_VEL
LIN {X 0,Y 275.47,Z 542.269,A -85,B 0,C 180,E1 -17372.93,E2 -17372.93} C_VEL
LIN {X 0,Y 275.49,Z 539.536,A -85,B 0,C 180,E1 -17375.193,E2 -17375.193} C_VEL
LIN {X 0,Y 275.597,Z 535.915,A -85,B 0,C 180,E1 -17377.331,E2 -17377.331} C_VEL
LIN {X 0,Y 275.894,Z 531.033,A -85,B 0,C 180,E1 -17379.536,E2 -17379.536} C_VEL
LIN {X 0,Y 276.382,Z 524.838,A -85,B 0,C 180,E1 -17381.743,E2 -17381.743} C_VEL
LIN {X 0,Y 277.424,Z 517.143,A -85,B 0,C 180,E1 -17383.931,E2 -17383.931} C_VEL
LIN {X 0,Y 278.384,Z 509.249,A -85,B 0,C 180,E1 -17385.752,E2 -17385.752} C_VEL
LIN {X 0,Y 279.018,Z 503.791,A -85,B 0,C 180,E1 -17386.829,E2 -17386.829} C_VEL
LIN {X 0,Y 280.388,Z 494.128,A -85,B 0,C 180,E1 -17388.453,E2 -17388.453} C_VEL
LIN {X 0,Y 281.448,Z 485.097,A -85,B 0,C 180,E1 -17389.706,E2 -17389.706} C_VEL
LIN {X 0,Y 280.67,Z 473.681,A -85,B 0,C 180,E1 -17391.084,E2 -17391.084} C_VEL
LIN {X 0,Y 279.302,Z 460.28,A -85,B 0,C 180,E1 -17392.375,E2 -17392.375} C_VEL
LIN {X 0,Y 277.675,Z 446.913,A -85,B 0,C 180,E1 -17393.372,E2 -17393.372} C_VEL
LIN {X 0,Y 276.617,Z 438.978,A -85,B 0,C 180,E1 -17393.841,E2 -17393.841} C_VEL
LIN {X 0,Y 277.316,Z 433.512,A -85,B 0,C 180,E1 -17397.499,E2 -17397.499} C_VEL
LIN {X 0,Y 278.414,Z 426.862,A -85,B 0,C 180,E1 -17402.017,E2 -17402.017} C_VEL
LIN {X 0,Y 279.304,Z 422.031,A -85,B 0,C 180,E1 -17405.367,E2 -17405.367} C_VEL
LIN {X 0,Y 279.507,Z 418.496,A -85,B 0,C 180,E1 -17407.913,E2 -17407.913} C_VEL
LIN {X 0,Y 278.873,Z 414.5,A -85,B 0,C 180,E1 -17410.943,E2 -17410.943} C_VEL
LIN {X 0,Y 277.885,Z 409.326,A -85,B 0,C 180,E1 -17415.09,E2 -17415.09} C_VEL
LIN {X 0,Y 277.263,Z 405.949,A -85,B 0,C 180,E1 -17418.016,E2 -17418.016} C_VEL
LIN {X 0,Y 277.271,Z 405.945,A -85,B 0,C 180,E1 -17422.53,E2 -17422.53} C_VEL
LIN {X 0,Y 277.263,Z 405.944,A -85,B 0,C 180,E1 -17426.105,E2 -17426.105} C_VEL
LIN {X 0,Y 277.28,Z 405.945,A -85,B 0,C 180,E1 -17429.54,E2 -17429.54} C_VEL
LIN {X 0,Y 277.31,Z 405.942,A -85,B 0,C 180,E1 -17432.858,E2 -17432.858} C_VEL
LIN {X 0,Y 277.3,Z 405.94,A -85,B 0,C 180,E1 -17436.076,E2 -17436.076} C_VEL
LIN {X 0,Y 277.302,Z 405.942,A -85,B 0,C 180,E1 -17440.762,E2 -17440.762} C_VEL
LIN {X 0,Y 277.426,Z 405.927,A -85,B 0,C 180,E1 -17445.324,E2 -17445.324} C_VEL
LIN {X 0,Y 277.472,Z 405.918,A -85,B 0,C 180,E1 -17449.786,E2 -17449.786} C_VEL
LIN {X 0,Y 277.632,Z 405.902,A -85,B 0,C 180,E1 -17452.727,E2 -17452.727} C_VEL
LIN {X 0,Y 277.833,Z 405.875,A -85,B 0,C 180,E1 -17458.549,E2 -17458.549} C_VEL
LIN {X 0,Y 277.828,Z 405.876,A -85,B 0,C 180,E1 -17461.448,E2 -17461.448} C_VEL
LIN {X 0,Y 277.615,Z 405.902,A -85,B 0,C 180,E1 -17467.271,E2 -17467.271} C_VEL
LIN {X 0,Y 277.47,Z 405.92,A -85,B 0,C 180,E1 -17470.211,E2 -17470.211} C_VEL
LIN {X 0,Y 277.423,Z 405.929,A -85,B 0,C 180,E1 -17474.673,E2 -17474.673} C_VEL
LIN {X 0,Y 277.299,Z 405.942,A -85,B 0,C 180,E1 -17479.236,E2 -17479.236} C_VEL
LIN {X 0,Y 277.309,Z 405.938,A -85,B 0,C 180,E1 -17483.921,E2 -17483.921} C_VEL
LIN {X 0,Y 277.33,Z 405.937,A -85,B 0,C 180,E1 -17487.499,E2 -17487.499} C_VEL
LIN {X 0,Y 277.26,Z 405.949,A -85,B 0,C 180,E1 -17490.469,E2 -17490.469} C_VEL
LIN {X 0,Y 277.257,Z 405.946,A -85,B 0,C 180,E1 -17493.892,E2 -17493.892} C_VEL
LIN {X 0,Y 277.272,Z 405.944,A -85,B 0,C 180,E1 -17497.467,E2 -17497.467} C_VEL
LIN {X 0,Y 277.218,Z 405.951,A -85,B 0,C 180,E1 -17501.233,E2 -17501.233} C_VEL
LIN {X 0,Y 277.209,Z 405.952,A -85,B 0,C 180,E1 -17505.223,E2 -17505.223} C_VEL
LIN {X 0,Y 277.225,Z 405.949,A -85,B 0,C 180,E1 -17509.509,E2 -17509.509} C_VEL
LIN {X 0,Y 277.271,Z 405.949,A -85,B 0,C 180,E1 -17512.526,E2 -17512.526} C_VEL
LIN {X 0,Y 277.252,Z 405.948,A -85,B 0,C 180,E1 -17516.1,E2 -17516.1} C_VEL
LIN {X 0,Y 277.266,Z 405.945,A -85,B 0,C 180,E1 -17519.534,E2 -17519.534} C_VEL
LIN {X 0,Y 277.36,Z 405.934,A -85,B 0,C 180,E1 -17522.859,E2 -17522.859} C_VEL
LIN {X 0,Y 277.331,Z 405.938,A -85,B 0,C 180,E1 -17526.075,E2 -17526.075} C_VEL
LIN {X 0,Y 277.346,Z 405.936,A -85,B 0,C 180,E1 -17530.761,E2 -17530.761} C_VEL
LIN {X 0,Y 277.434,Z 405.923,A -85,B 0,C 180,E1 -17535.321,E2 -17535.321} C_VEL
LIN {X 0,Y 277.458,Z 405.922,A -85,B 0,C 180,E1 -17539.782,E2 -17539.782} C_VEL
LIN {X 0,Y 277.637,Z 405.899,A -85,B 0,C 180,E1 -17542.724,E2 -17542.724} C_VEL
LIN {X 0,Y 277.814,Z 405.878,A -85,B 0,C 180,E1 -17548.545,E2 -17548.545} C_VEL
LIN {X 0,Y 277.814,Z 405.876,A -85,B 0,C 180,E1 -17551.444,E2 -17551.444} C_VEL
LIN {X 0,Y 277.643,Z 405.897,A -85,B 0,C 180,E1 -17557.266,E2 -17557.266} C_VEL
LIN {X 0,Y 277.496,Z 405.92,A -85,B 0,C 180,E1 -17560.206,E2 -17560.206} C_VEL
LIN {X 0,Y 277.421,Z 405.926,A -85,B 0,C 180,E1 -17564.669,E2 -17564.669} C_VEL
LIN {X 0,Y 277.329,Z 405.937,A -85,B 0,C 180,E1 -17569.229,E2 -17569.229} C_VEL
LIN {X 0,Y 277.258,Z 405.95,A -85,B 0,C 180,E1 -17573.92,E2 -17573.92} C_VEL
LIN {X 0,Y 277.069,Z 405.97,A -85,B 0,C 180,E1 -17577.406,E2 -17577.406} C_VEL
LIN {X 0,Y 276.677,Z 406.019,A -85,B 0,C 180,E1 -17580.525,E2 -17580.525} C_VEL
LIN {X 0,Y 276.2,Z 406.085,A -85,B 0,C 180,E1 -17584.034,E2 -17584.034} C_VEL
LIN {X 0,Y 276.091,Z 407.029,A -85,B 0,C 180,E1 -17585.829,E2 -17585.829} C_VEL
LIN {X 0,Y 276.016,Z 409.041,A -85,B 0,C 180,E1 -17588.313,E2 -17588.313} C_VEL
LIN {X 0,Y 279.365,Z 423.071,A -85,B 0,C 180,E1 -17589.341,E2 -17589.341} C_VEL
LIN {X 0,Y 282.093,Z 435.722,A -85,B 0,C 180,E1 -17590.531,E2 -17590.531} C_VEL
LIN {X 0,Y 283.624,Z 444.099,A -85,B 0,C 180,E1 -17591.477,E2 -17591.477} C_VEL
LIN {X 0,Y 282.405,Z 455.083,A -85,B 0,C 180,E1 -17592.767,E2 -17592.767} C_VEL
LIN {X 0,Y 280.956,Z 466.484,A -85,B 0,C 180,E1 -17594.451,E2 -17594.451} C_VEL
LIN {X 0,Y 279.618,Z 476.99,A -85,B 0,C 180,E1 -17596.393,E2 -17596.393} C_VEL
LIN {X 0,Y 278.33,Z 486.07,A -85,B 0,C 180,E1 -17598.486,E2 -17598.486} C_VEL
LIN {X 0,Y 277.332,Z 493.735,A -85,B 0,C 180,E1 -17600.69,E2 -17600.69} C_VEL
LIN {X 0,Y 276.584,Z 499.85,A -85,B 0,C 180,E1 -17602.882,E2 -17602.882} C_VEL
LIN {X 0,Y 276.034,Z 504.984,A -85,B 0,C 180,E1 -17605.22,E2 -17605.22} C_VEL
LIN {X 0,Y 275.591,Z 508.919,A -85,B 0,C 180,E1 -17607.622,E2 -17607.622} C_VEL
LIN {X 0,Y 275.325,Z 511.8,A -85,B 0,C 180,E1 -17610.2,E2 -17610.2} C_VEL
LIN {X 0,Y 275.34,Z 513.595,A -85,B 0,C 180,E1 -17613.284,E2 -17613.284} C_VEL
LIN {X 0,Y 275.692,Z 513.67,A -85,B 0,C 180,E1 -17615.93,E2 -17615.93} C_VEL
LIN {X 0,Y 276.075,Z 513.081,A -85,B 0,C 180,E1 -17617.553,E2 -17617.553} C_VEL
LIN {X 0,Y 276.863,Z 511.346,A -85,B 0,C 180,E1 -17619.901,E2 -17619.901} C_VEL
LIN {X 0,Y 277.881,Z 508.432,A -85,B 0,C 180,E1 -17622.334,E2 -17622.334} C_VEL
LIN {X 0,Y 279.234,Z 504.408,A -85,B 0,C 180,E1 -17624.678,E2 -17624.678} C_VEL
LIN {X 0,Y 281.096,Z 498.654,A -85,B 0,C 180,E1 -17627.151,E2 -17627.151} C_VEL
LIN {X 0,Y 283.399,Z 491.099,A -85,B 0,C 180,E1 -17629.644,E2 -17629.644} C_VEL
LIN {X 0,Y 285.977,Z 482.322,A -85,B 0,C 180,E1 -17631.878,E2 -17631.878} C_VEL
LIN {X 0,Y 288.319,Z 473.404,A -85,B 0,C 180,E1 -17633.704,E2 -17633.704} C_VEL
LIN {X 0,Y 290.759,Z 463.215,A -85,B 0,C 180,E1 -17635.376,E2 -17635.376} C_VEL
LIN {X 0,Y 292.343,Z 455.618,A -85,B 0,C 180,E1 -17636.412,E2 -17636.412} C_VEL
LIN {X 0,Y 290.499,Z 445.114,A -85,B 0,C 180,E1 -17638.197,E2 -17638.197} C_VEL
LIN {X 0,Y 287.692,Z 436.489,A -85,B 0,C 180,E1 -17639.696,E2 -17639.696} C_VEL
LIN {X 0,Y 283.141,Z 424.832,A -85,B 0,C 180,E1 -17641.693,E2 -17641.693} C_VEL
LIN {X 0,Y 281.527,Z 421.503,A -85,B 0,C 180,E1 -17642.291,E2 -17642.291} C_VEL
LIN {X 0,Y 280.183,Z 418.924,A -85,B 0,C 180,E1 -17642.755,E2 -17642.755} C_VEL
LIN {X 0,Y 278.467,Z 415.996,A -85,B 0,C 180,E1 -17643.347,E2 -17643.347} C_VEL
LIN {X 0,Y 278.15,Z 414.799,A -85,B 0,C 180,E1 -17643.532,E2 -17643.532} C_VEL
LIN {X 0,Y 278.199,Z 414.424,A -85,B 0,C 180,E1 -17644.393,E2 -17644.393} C_VEL
LIN {X 0,Y 277.625,Z 414.047,A -85,B 0,C 180,E1 -17645.601,E2 -17645.601} C_VEL
LIN {X 0,Y 274.975,Z 413.837,A -85,B 0,C 180,E1 -17647.58,E2 -17647.58} C_VEL
LIN {X 0,Y 271.842,Z 413.695,A -85,B 0,C 180,E1 -17650.011,E2 -17650.011} C_VEL
LIN {X 0,Y 271.471,Z 413.531,A -85,B 0,C 180,E1 -17650.849,E2 -17650.849} C_VEL
LIN {X 0,Y 271.333,Z 412.624,A -85,B 0,C 180,E1 -17655.013,E2 -17655.013} C_VEL
LIN {X 0,Y 271.176,Z 412.091,A -85,B 0,C 180,E1 -17659.691,E2 -17659.691} C_VEL
LIN {X 0,Y 271.24,Z 412.166,A -85,B 0,C 180,E1 -17664.494,E2 -17664.494} C_VEL
LIN {X 0,Y 271.283,Z 412.708,A -85,B 0,C 180,E1 -17668.273,E2 -17668.273} C_VEL
LIN {X 0,Y 271.393,Z 413.477,A -85,B 0,C 180,E1 -17671.302,E2 -17671.302} C_VEL
LIN {X 0,Y 271.591,Z 414.694,A -85,B 0,C 180,E1 -17674.703,E2 -17674.703} C_VEL
LIN {X 0,Y 271.909,Z 416.409,A -85,B 0,C 180,E1 -17678.341,E2 -17678.341} C_VEL
LIN {X 0,Y 272.342,Z 418.713,A -85,B 0,C 180,E1 -17682.142,E2 -17682.142} C_VEL
LIN {X 0,Y 272.854,Z 421.686,A -85,B 0,C 180,E1 -17686.156,E2 -17686.156} C_VEL
LIN {X 0,Y 273.314,Z 425.083,A -85,B 0,C 180,E1 -17690.004,E2 -17690.004} C_VEL
LIN {X 0,Y 273.451,Z 427.922,A -85,B 0,C 180,E1 -17692.821,E2 -17692.821} C_VEL
LIN {X 0,Y 272.788,Z 431.031,A -85,B 0,C 180,E1 -17695.533,E2 -17695.533} C_VEL
LIN {X 0,Y 272.235,Z 433.011,A -85,B 0,C 180,E1 -17697.152,E2 -17697.152} C_VEL
LIN {X 0,Y 273.142,Z 436.455,A -85,B 0,C 180,E1 -17697.595,E2 -17697.595} C_VEL
LIN {X 0,Y 274.116,Z 438.754,A -85,B 0,C 180,E1 -17697.984,E2 -17697.984} C_VEL
LIN {X 0,Y 278.088,Z 451.547,A -85,B 0,C 180,E1 -17699.882,E2 -17699.882} C_VEL
LIN {X 0,Y 280.51,Z 463.236,A -85,B 0,C 180,E1 -17701.58,E2 -17701.58} C_VEL
LIN {X 0,Y 281.711,Z 473.826,A -85,B 0,C 180,E1 -17703.124,E2 -17703.124} C_VEL
LIN {X 0,Y 281.868,Z 483.671,A -85,B 0,C 180,E1 -17704.635,E2 -17704.635} C_VEL
LIN {X 0,Y 280.911,Z 494.42,A -85,B 0,C 180,E1 -17706.41,E2 -17706.41} C_VEL
LIN {X 0,Y 278.315,Z 504.106,A -85,B 0,C 180,E1 -17708.139,E2 -17708.139} C_VEL
LIN {X 0,Y 275.501,Z 513.7,A -85,B 0,C 180,E1 -17710.251,E2 -17710.251} C_VEL
LIN {X 0,Y 273.279,Z 521.525,A -85,B 0,C 180,E1 -17712.418,E2 -17712.418} C_VEL
LIN {X 0,Y 271.956,Z 526.943,A -85,B 0,C 180,E1 -17714.262,E2 -17714.262} C_VEL
LIN {X 0,Y 270.323,Z 532.355,A -85,B 0,C 180,E1 -17716.474,E2 -17716.474} C_VEL
LIN {X 0,Y 269.298,Z 536.638,A -85,B 0,C 180,E1 -17718.719,E2 -17718.719} C_VEL
LIN {X 0,Y 268.673,Z 539.902,A -85,B 0,C 180,E1 -17720.976,E2 -17720.976} C_VEL
LIN {X 0,Y 268.403,Z 541.573,A -85,B 0,C 180,E1 -17722.483,E2 -17722.483} C_VEL
LIN {X 0,Y 268.245,Z 543.21,A -85,B 0,C 180,E1 -17724.632,E2 -17724.632} C_VEL
LIN {X 0,Y 268.332,Z 544.081,A -85,B 0,C 180,E1 -17727.003,E2 -17727.003} C_VEL
LIN {X 0,Y 268.374,Z 544.124,A -85,B 0,C 180,E1 -17728.505,E2 -17728.505} C_VEL
LIN {X 0,Y 268.553,Z 543.729,A -85,B 0,C 180,E1 -17730.005,E2 -17730.005} C_VEL
LIN {X 0,Y 268.442,Z 542.891,A -85,B 0,C 180,E1 -17731.506,E2 -17731.506} C_VEL
LIN {X 0,Y 268.399,Z 541.643,A -85,B 0,C 180,E1 -17733.007,E2 -17733.007} C_VEL
LIN {X 0,Y 268.429,Z 539.966,A -85,B 0,C 180,E1 -17734.51,E2 -17734.51} C_VEL
LIN {X 0,Y 268.495,Z 536.529,A -85,B 0,C 180,E1 -17736.77,E2 -17736.77} C_VEL
LIN {X 0,Y 268.718,Z 531.948,A -85,B 0,C 180,E1 -17739.034,E2 -17739.034} C_VEL
LIN {X 0,Y 269.271,Z 524.959,A -85,B 0,C 180,E1 -17741.675,E2 -17741.675} C_VEL
LIN {X 0,Y 270.293,Z 517.42,A -85,B 0,C 180,E1 -17743.922,E2 -17743.922} C_VEL
LIN {X 0,Y 271.294,Z 509.704,A -85,B 0,C 180,E1 -17745.789,E2 -17745.789} C_VEL
LIN {X 0,Y 272.018,Z 503.453,A -85,B 0,C 180,E1 -17747.066,E2 -17747.066} C_VEL
LIN {X 0,Y 273.437,Z 493.713,A -85,B 0,C 180,E1 -17748.745,E2 -17748.745} C_VEL
LIN {X 0,Y 274.43,Z 486.081,A -85,B 0,C 180,E1 -17749.841,E2 -17749.841} C_VEL
LIN {X 0,Y 273.61,Z 473.62,A -85,B 0,C 180,E1 -17751.411,E2 -17751.411} C_VEL
LIN {X 0,Y 272.383,Z 461.227,A -85,B 0,C 180,E1 -17752.652,E2 -17752.652} C_VEL
LIN {X 0,Y 270.754,Z 447.482,A -85,B 0,C 180,E1 -17753.724,E2 -17753.724} C_VEL
LIN {X 0,Y 269.587,Z 438.642,A -85,B 0,C 180,E1 -17754.255,E2 -17754.255} C_VEL
LIN {X 0,Y 270.509,Z 432.171,A -85,B 0,C 180,E1 -17758.733,E2 -17758.733} C_VEL
LIN {X 0,Y 271.58,Z 426.21,A -85,B 0,C 180,E1 -17762.923,E2 -17762.923} C_VEL
LIN {X 0,Y 272.449,Z 421.366,A -85,B 0,C 180,E1 -17766.397,E2 -17766.397} C_VEL
LIN {X 0,Y 272.186,Z 417.631,A -85,B 0,C 180,E1 -17769.228,E2 -17769.228} C_VEL
LIN {X 0,Y 271.495,Z 413.762,A -85,B 0,C 180,E1 -17772.308,E2 -17772.308} C_VEL
LIN {X 0,Y 270.548,Z 408.539,A -85,B 0,C 180,E1 -17776.671,E2 -17776.671} C_VEL
LIN {X 0,Y 270.208,Z 406.827,A -85,B 0,C 180,E1 -17778.282,E2 -17778.282} C_VEL
LIN {X 0,Y 270.225,Z 406.825,A -85,B 0,C 180,E1 -17781.376,E2 -17781.376} C_VEL
LIN {X 0,Y 270.215,Z 406.826,A -85,B 0,C 180,E1 -17785.095,E2 -17785.095} C_VEL
LIN {X 0,Y 270.202,Z 406.83,A -85,B 0,C 180,E1 -17789.138,E2 -17789.138} C_VEL
LIN {X 0,Y 270.241,Z 406.819,A -85,B 0,C 180,E1 -17792.164,E2 -17792.164} C_VEL
LIN {X 0,Y 270.246,Z 406.821,A -85,B 0,C 180,E1 -17795.543,E2 -17795.543} C_VEL
LIN {X 0,Y 270.241,Z 406.819,A -85,B 0,C 180,E1 -17800.239,E2 -17800.239} C_VEL
LIN {X 0,Y 270.386,Z 406.806,A -85,B 0,C 180,E1 -17804.933,E2 -17804.933} C_VEL
LIN {X 0,Y 270.424,Z 406.797,A -85,B 0,C 180,E1 -17809.517,E2 -17809.517} C_VEL
LIN {X 0,Y 270.591,Z 406.778,A -85,B 0,C 180,E1 -17812.537,E2 -17812.537} C_VEL
LIN {X 0,Y 270.799,Z 406.751,A -85,B 0,C 180,E1 -17818.512,E2 -17818.512} C_VEL
LIN {X 0,Y 270.793,Z 406.752,A -85,B 0,C 180,E1 -17821.486,E2 -17821.486} C_VEL
LIN {X 0,Y 270.577,Z 406.778,A -85,B 0,C 180,E1 -17827.461,E2 -17827.461} C_VEL
LIN {X 0,Y 270.421,Z 406.8,A -85,B 0,C 180,E1 -17830.48,E2 -17830.48} C_VEL
LIN {X 0,Y 270.382,Z 406.804,A -85,B 0,C 180,E1 -17835.064,E2 -17835.064} C_VEL
LIN {X 0,Y 270.238,Z 406.82,A -85,B 0,C 180,E1 -17839.759,E2 -17839.759} C_VEL
LIN {X 0,Y 270.25,Z 406.821,A -85,B 0,C 180,E1 -17844.586,E2 -17844.586} C_VEL
LIN {X 0,Y 270.257,Z 406.818,A -85,B 0,C 180,E1 -17847.909,E2 -17847.909} C_VEL
LIN {X 0,Y 270.185,Z 406.826,A -85,B 0,C 180,E1 -17851.346,E2 -17851.346} C_VEL
LIN {X 0,Y 270.211,Z 406.826,A -85,B 0,C 180,E1 -17854.902,E2 -17854.902} C_VEL
LIN {X 0,Y 270.208,Z 406.827,A -85,B 0,C 180,E1 -17858.707,E2 -17858.707} C_VEL
LIN {X 0,Y 270.174,Z 406.829,A -85,B 0,C 180,E1 -17863.245,E2 -17863.245} C_VEL
LIN {X 0,Y 270.171,Z 406.828,A -85,B 0,C 180,E1 -17867.436,E2 -17867.436} C_VEL
LIN {X 0,Y 270.214,Z 406.823,A -85,B 0,C 180,E1 -17871.37,E2 -17871.37} C_VEL
LIN {X 0,Y 270.207,Z 406.824,A -85,B 0,C 180,E1 -17875.09,E2 -17875.09} C_VEL
LIN {X 0,Y 270.205,Z 406.825,A -85,B 0,C 180,E1 -17879.126,E2 -17879.126} C_VEL
LIN {X 0,Y 270.267,Z 406.82,A -85,B 0,C 180,E1 -17882.142,E2 -17882.142} C_VEL
LIN {X 0,Y 270.28,Z 406.814,A -85,B 0,C 180,E1 -17885.514,E2 -17885.514} C_VEL
LIN {X 0,Y 270.303,Z 406.816,A -85,B 0,C 180,E1 -17890.239,E2 -17890.239} C_VEL
LIN {X 0,Y 270.402,Z 406.8,A -85,B 0,C 180,E1 -17894.93,E2 -17894.93} C_VEL
LIN {X 0,Y 270.41,Z 406.799,A -85,B 0,C 180,E1 -17899.513,E2 -17899.513} C_VEL
LIN {X 0,Y 270.595,Z 406.777,A -85,B 0,C 180,E1 -17902.533,E2 -17902.533} C_VEL
LIN {X 0,Y 270.78,Z 406.754,A -85,B 0,C 180,E1 -17908.507,E2 -17908.507} C_VEL
LIN {X 0,Y 270.78,Z 406.752,A -85,B 0,C 180,E1 -17911.482,E2 -17911.482} C_VEL
LIN {X 0,Y 270.601,Z 406.775,A -85,B 0,C 180,E1 -17917.456,E2 -17917.456} C_VEL
LIN {X 0,Y 270.431,Z 406.798,A -85,B 0,C 180,E1 -17920.476,E2 -17920.476} C_VEL
LIN {X 0,Y 270.389,Z 406.801,A -85,B 0,C 180,E1 -17925.059,E2 -17925.059} C_VEL
LIN {X 0,Y 270.285,Z 406.817,A -85,B 0,C 180,E1 -17929.75,E2 -17929.75} C_VEL
LIN {X 0,Y 270.161,Z 406.831,A -85,B 0,C 180,E1 -17934.59,E2 -17934.59} C_VEL
LIN {X 0,Y 269.958,Z 406.86,A -85,B 0,C 180,E1 -17937.937,E2 -17937.937} C_VEL
LIN {X 0,Y 269.491,Z 406.915,A -85,B 0,C 180,E1 -17941.43,E2 -17941.43} C_VEL
LIN {X 0,Y 269.046,Z 407.174,A -85,B 0,C 180,E1 -17945.069,E2 -17945.069} C_VEL
LIN {X 0,Y 268.984,Z 409.419,A -85,B 0,C 180,E1 -17947.88,E2 -17947.88} C_VEL
LIN {X 0,Y 272.369,Z 423.652,A -85,B 0,C 180,E1 -17948.965,E2 -17948.965} C_VEL
LIN {X 0,Y 275.034,Z 436.183,A -85,B 0,C 180,E1 -17950.174,E2 -17950.174} C_VEL
LIN {X 0,Y 276.693,Z 445.027,A -85,B 0,C 180,E1 -17951.201,E2 -17951.201} C_VEL
LIN {X 0,Y 275.435,Z 455.783,A -85,B 0,C 180,E1 -17952.508,E2 -17952.508} C_VEL
LIN {X 0,Y 274.062,Z 466.378,A -85,B 0,C 180,E1 -17954.11,E2 -17954.11} C_VEL
LIN {X 0,Y 272.588,Z 477.447,A -85,B 0,C 180,E1 -17956.203,E2 -17956.203} C_VEL
LIN {X 0,Y 271.305,Z 486.263,A -85,B 0,C 180,E1 -17958.285,E2 -17958.285} C_VEL
LIN {X 0,Y 270.331,Z 493.639,A -85,B 0,C 180,E1 -17960.439,E2 -17960.439} C_VEL
LIN {X 0,Y 269.541,Z 499.851,A -85,B 0,C 180,E1 -17962.685,E2 -17962.685} C_VEL
LIN {X 0,Y 268.988,Z 504.749,A -85,B 0,C 180,E1 -17964.916,E2 -17964.916} C_VEL
LIN {X 0,Y 268.515,Z 509.232,A -85,B 0,C 180,E1 -17967.625,E2 -17967.625} C_VEL
LIN {X 0,Y 268.234,Z 512.055,A -85,B 0,C 180,E1 -17970.146,E2 -17970.146} C_VEL
LIN {X 0,Y 268.228,Z 513.829,A -85,B 0,C 180,E1 -17972.965,E2 -17972.965} C_VEL
LIN {X 0,Y 268.501,Z 514.227,A -85,B 0,C 180,E1 -17975.243,E2 -17975.243} C_VEL
LIN {X 0,Y 268.856,Z 513.956,A -85,B 0,C 180,E1 -17976.916,E2 -17976.916} C_VEL
LIN {X 0,Y 269.702,Z 512.35,A -85,B 0,C 180,E1 -17979.714,E2 -17979.714} C_VEL
LIN {X 0,Y 270.963,Z 509.13,A -85,B 0,C 180,E1 -17982.648,E2 -17982.648} C_VEL
LIN {X 0,Y 272.401,Z 505.199,A -85,B 0,C 180,E1 -17985.05,E2 -17985.05} C_VEL
LIN {X 0,Y 274.429,Z 499.45,A -85,B 0,C 180,E1 -17987.638,E2 -17987.638} C_VEL
LIN {X 0,Y 276.748,Z 492.371,A -85,B 0,C 180,E1 -17990.079,E2 -17990.079} C_VEL
LIN {X 0,Y 279.087,Z 485.148,A -85,B 0,C 180,E1 -17992.04,E2 -17992.04} C_VEL
LIN {X 0,Y 281.445,Z 476.742,A -85,B 0,C 180,E1 -17993.909,E2 -17993.909} C_VEL
LIN {X 0,Y 284.49,Z 465.216,A -85,B 0,C 180,E1 -17995.929,E2 -17995.929} C_VEL
LIN {X 0,Y 286.195,Z 457.701,A -85,B 0,C 180,E1 -17997.01,E2 -17997.01} C_VEL
LIN {X 0,Y 284.542,Z 447.723,A -85,B 0,C 180,E1 -17998.815,E2 -17998.815} C_VEL
LIN {X 0,Y 280.742,Z 435.721,A -85,B 0,C 180,E1 -18001.044,E2 -18001.044} C_VEL
LIN {X 0,Y 277.313,Z 427.053,A -85,B 0,C 180,E1 -18002.645,E2 -18002.645} C_VEL
LIN {X 0,Y 275.414,Z 423.463,A -85,B 0,C 180,E1 -18003.39,E2 -18003.39} C_VEL
LIN {X 0,Y 273.437,Z 419.841,A -85,B 0,C 180,E1 -18004.147,E2 -18004.147} C_VEL
LIN {X 0,Y 271.644,Z 416.907,A -85,B 0,C 180,E1 -18004.801,E2 -18004.801} C_VEL
LIN {X 0,Y 271.294,Z 415.518,A -85,B 0,C 180,E1 -18005.017,E2 -18005.017} C_VEL
LIN {X 0,Y 271.532,Z 414.574,A -85,B 0,C 180,E1 -18007.437,E2 -18007.437} C_VEL
LIN {X 0,Y 271.471,Z 413.531,A -85,B 0,C 180,E1 -18010.849,E2 -18010.849} C_VEL
LIN {X 0,Y 270.716,Z 413.376,A -85,B 0,C 180,E1 -18012.085,E2 -18012.085} C_VEL
LIN {X 0,Y 267.845,Z 413.561,A -85,B 0,C 180,E1 -18014.103,E2 -18014.103} C_VEL
LIN {X 0,Y 265.444,Z 413.813,A -85,B 0,C 180,E1 -18015.743,E2 -18015.743} C_VEL
LIN {X 0,Y 264.393,Z 413.88,A -85,B 0,C 180,E1 -18017.013,E2 -18017.013} C_VEL
LIN {X 0,Y 264.292,Z 413.857,A -85,B 0,C 180,E1 -18017.444,E2 -18017.444} C_VEL
LIN {X 0,Y 264.252,Z 413.664,A -85,B 0,C 180,E1 -18021.861,E2 -18021.861} C_VEL
LIN {X 0,Y 264.321,Z 413.885,A -85,B 0,C 180,E1 -18025.325,E2 -18025.325} C_VEL
LIN {X 0,Y 264.402,Z 414.455,A -85,B 0,C 180,E1 -18028.713,E2 -18028.713} C_VEL
LIN {X 0,Y 264.496,Z 415.388,A -85,B 0,C 180,E1 -18032.103,E2 -18032.103} C_VEL
LIN {X 0,Y 264.746,Z 416.765,A -85,B 0,C 180,E1 -18035.735,E2 -18035.735} C_VEL
LIN {X 0,Y 265.16,Z 418.834,A -85,B 0,C 180,E1 -18039.779,E2 -18039.779} C_VEL
LIN {X 0,Y 265.553,Z 421.201,A -85,B 0,C 180,E1 -18043.482,E2 -18043.482} C_VEL
LIN {X 0,Y 265.955,Z 423.555,A -85,B 0,C 180,E1 -18046.611,E2 -18046.611} C_VEL
LIN {X 0,Y 266.418,Z 427.177,A -85,B 0,C 180,E1 -18050.729,E2 -18050.729} C_VEL
LIN {X 0,Y 266.47,Z 429.093,A -85,B 0,C 180,E1 -18052.663,E2 -18052.663} C_VEL
LIN {X 0,Y 265.833,Z 432.085,A -85,B 0,C 180,E1 -18055.368,E2 -18055.368} C_VEL
LIN {X 0,Y 265.76,Z 432.522,A -85,B 0,C 180,E1 -18055.611,E2 -18055.611} C_VEL
LIN {X 0,Y 266.778,Z 436.056,A -85,B 0,C 180,E1 -18056.136,E2 -18056.136} C_VEL
LIN {X 0,Y 267.652,Z 438.039,A -85,B 0,C 180,E1 -18056.511,E2 -18056.511} C_VEL
LIN {X 0,Y 269.066,Z 442.034,A -85,B 0,C 180,E1 -18057.167,E2 -18057.167} C_VEL
LIN {X 0,Y 272.787,Z 455.341,A -85,B 0,C 180,E1 -18059.302,E2 -18059.302} C_VEL
LIN {X 0,Y 274.827,Z 466.857,A -85,B 0,C 180,E1 -18061.081,E2 -18061.081} C_VEL
LIN {X 0,Y 275.633,Z 477.014,A -85,B 0,C 180,E1 -18062.687,E2 -18062.687} C_VEL
LIN {X 0,Y 275.489,Z 486.889,A -85,B 0,C 180,E1 -18064.305,E2 -18064.305} C_VEL
LIN {X 0,Y 274.493,Z 495.494,A -85,B 0,C 180,E1 -18065.823,E2 -18065.823} C_VEL
LIN {X 0,Y 271.796,Z 504.864,A -85,B 0,C 180,E1 -18067.586,E2 -18067.586} C_VEL
LIN {X 0,Y 268.869,Z 514.229,A -85,B 0,C 180,E1 -18069.743,E2 -18069.743} C_VEL
LIN {X 0,Y 266.509,Z 521.882,A -85,B 0,C 180,E1 -18071.968,E2 -18071.968} C_VEL
LIN {X 0,Y 265.132,Z 527.154,A -85,B 0,C 180,E1 -18073.846,E2 -18073.846} C_VEL
LIN {X 0,Y 263.423,Z 532.397,A -85,B 0,C 180,E1 -18076.113,E2 -18076.113} C_VEL
LIN {X 0,Y 262.309,Z 536.572,A -85,B 0,C 180,E1 -18078.414,E2 -18078.414} C_VEL
LIN {X 0,Y 261.616,Z 539.747,A -85,B 0,C 180,E1 -18080.73,E2 -18080.73} C_VEL
LIN {X 0,Y 261.218,Z 542.496,A -85,B 0,C 180,E1 -18083.828,E2 -18083.828} C_VEL
LIN {X 0,Y 261.257,Z 543.68,A -85,B 0,C 180,E1 -18086.922,E2 -18086.922} C_VEL
LIN {X 0,Y 261.293,Z 543.648,A -85,B 0,C 180,E1 -18088.464,E2 -18088.464} C_VEL
LIN {X 0,Y 261.469,Z 543.194,A -85,B 0,C 180,E1 -18090.006,E2 -18090.006} C_VEL
LIN {X 0,Y 261.358,Z 542.312,A -85,B 0,C 180,E1 -18091.546,E2 -18091.546} C_VEL
LIN {X 0,Y 261.329,Z 541.019,A -85,B 0,C 180,E1 -18093.089,E2 -18093.089} C_VEL
LIN {X 0,Y 261.389,Z 537.571,A -85,B 0,C 180,E1 -18095.822,E2 -18095.822} C_VEL
LIN {X 0,Y 261.569,Z 532.702,A -85,B 0,C 180,E1 -18098.504,E2 -18098.504} C_VEL
LIN {X 0,Y 261.978,Z 527.174,A -85,B 0,C 180,E1 -18100.829,E2 -18100.829} C_VEL
LIN {X 0,Y 262.794,Z 520.263,A -85,B 0,C 180,E1 -18103.145,E2 -18103.145} C_VEL
LIN {X 0,Y 263.939,Z 511.596,A -85,B 0,C 180,E1 -18105.448,E2 -18105.448} C_VEL
LIN {X 0,Y 264.746,Z 504.651,A -85,B 0,C 180,E1 -18106.983,E2 -18106.983} C_VEL
LIN {X 0,Y 266.376,Z 494.29,A -85,B 0,C 180,E1 -18108.862,E2 -18108.862} C_VEL
LIN {X 0,Y 267.362,Z 486.866,A -85,B 0,C 180,E1 -18109.987,E2 -18109.987} C_VEL
LIN {X 0,Y 266.773,Z 475.869,A -85,B 0,C 180,E1 -18111.445,E2 -18111.445} C_VEL
LIN {X 0,Y 265.713,Z 464.109,A -85,B 0,C 180,E1 -18112.731,E2 -18112.731} C_VEL
LIN {X 0,Y 264.172,Z 450.789,A -85,B 0,C 180,E1 -18113.883,E2 -18113.883} C_VEL
LIN {X 0,Y 262.575,Z 438.289,A -85,B 0,C 180,E1 -18114.705,E2 -18114.705} C_VEL
LIN {X 0,Y 263.399,Z 432.665,A -85,B 0,C 180,E1 -18118.709,E2 -18118.709} C_VEL
LIN {X 0,Y 264.528,Z 426.726,A -85,B 0,C 180,E1 -18123.006,E2 -18123.006} C_VEL
LIN {X 0,Y 265.402,Z 421.984,A -85,B 0,C 180,E1 -18126.512,E2 -18126.512} C_VEL
LIN {X 0,Y 265.302,Z 419.413,A -85,B 0,C 180,E1 -18128.507,E2 -18128.507} C_VEL
LIN {X 0,Y 264.542,Z 415.174,A -85,B 0,C 180,E1 -18131.937,E2 -18131.937} C_VEL
LIN {X 0,Y 263.635,Z 410.256,A -85,B 0,C 180,E1 -18136.122,E2 -18136.122} C_VEL
LIN {X 0,Y 263.155,Z 407.707,A -85,B 0,C 180,E1 -18138.405,E2 -18138.405} C_VEL
LIN {X 0,Y 263.193,Z 407.701,A -85,B 0,C 180,E1 -18143.241,E2 -18143.241} C_VEL
LIN {X 0,Y 263.146,Z 407.705,A -85,B 0,C 180,E1 -18147.712,E2 -18147.712} C_VEL
LIN {X 0,Y 263.166,Z 407.701,A -85,B 0,C 180,E1 -18151.806,E2 -18151.806} C_VEL
LIN {X 0,Y 263.208,Z 407.7,A -85,B 0,C 180,E1 -18155.219,E2 -18155.219} C_VEL
LIN {X 0,Y 263.227,Z 407.694,A -85,B 0,C 180,E1 -18159.689,E2 -18159.689} C_VEL
LIN {X 0,Y 263.328,Z 407.682,A -85,B 0,C 180,E1 -18164.519,E2 -18164.519} C_VEL
LIN {X 0,Y 263.363,Z 407.678,A -85,B 0,C 180,E1 -18169.233,E2 -18169.233} C_VEL
LIN {X 0,Y 263.553,Z 407.653,A -85,B 0,C 180,E1 -18172.337,E2 -18172.337} C_VEL
LIN {X 0,Y 263.764,Z 407.627,A -85,B 0,C 180,E1 -18178.472,E2 -18178.472} C_VEL
LIN {X 0,Y 263.756,Z 407.628,A -85,B 0,C 180,E1 -18181.526,E2 -18181.526} C_VEL
LIN {X 0,Y 263.541,Z 407.654,A -85,B 0,C 180,E1 -18187.661,E2 -18187.661} C_VEL
LIN {X 0,Y 263.361,Z 407.681,A -85,B 0,C 180,E1 -18190.765,E2 -18190.765} C_VEL
LIN {X 0,Y 263.325,Z 407.681,A -85,B 0,C 180,E1 -18195.478,E2 -18195.478} C_VEL
LIN {X 0,Y 263.223,Z 407.696,A -85,B 0,C 180,E1 -18200.308,E2 -18200.308} C_VEL
LIN {X 0,Y 263.204,Z 407.697,A -85,B 0,C 180,E1 -18205.29,E2 -18205.29} C_VEL
LIN {X 0,Y 263.167,Z 407.705,A -85,B 0,C 180,E1 -18208.729,E2 -18208.729} C_VEL
LIN {X 0,Y 263.14,Z 407.705,A -85,B 0,C 180,E1 -18212.285,E2 -18212.285} C_VEL
LIN {X 0,Y 263.19,Z 407.702,A -85,B 0,C 180,E1 -18216.759,E2 -18216.759} C_VEL
LIN {X 0,Y 263.115,Z 407.707,A -85,B 0,C 180,E1 -18219.869,E2 -18219.869} C_VEL
LIN {X 0,Y 263.112,Z 407.709,A -85,B 0,C 180,E1 -18223.984,E2 -18223.984} C_VEL
LIN {X 0,Y 263.127,Z 407.709,A -85,B 0,C 180,E1 -18228.403,E2 -18228.403} C_VEL
LIN {X 0,Y 263.165,Z 407.703,A -85,B 0,C 180,E1 -18232.098,E2 -18232.098} C_VEL
LIN {X 0,Y 263.157,Z 407.703,A -85,B 0,C 180,E1 -18235.881,E2 -18235.881} C_VEL
LIN {X 0,Y 263.152,Z 407.703,A -85,B 0,C 180,E1 -18239.502,E2 -18239.502} C_VEL
LIN {X 0,Y 263.195,Z 407.698,A -85,B 0,C 180,E1 -18242.998,E2 -18242.998} C_VEL
LIN {X 0,Y 263.189,Z 407.702,A -85,B 0,C 180,E1 -18246.382,E2 -18246.382} C_VEL
LIN {X 0,Y 263.266,Z 407.69,A -85,B 0,C 180,E1 -18249.688,E2 -18249.688} C_VEL
LIN {X 0,Y 263.35,Z 407.681,A -85,B 0,C 180,E1 -18254.517,E2 -18254.517} C_VEL
LIN {X 0,Y 263.353,Z 407.678,A -85,B 0,C 180,E1 -18259.228,E2 -18259.228} C_VEL
LIN {X 0,Y 263.554,Z 407.656,A -85,B 0,C 180,E1 -18262.332,E2 -18262.332} C_VEL
LIN {X 0,Y 263.744,Z 407.631,A -85,B 0,C 180,E1 -18268.468,E2 -18268.468} C_VEL
LIN {X 0,Y 263.744,Z 407.629,A -85,B 0,C 180,E1 -18271.521,E2 -18271.521} C_VEL
LIN {X 0,Y 263.563,Z 407.653,A -85,B 0,C 180,E1 -18277.656,E2 -18277.656} C_VEL
LIN {X 0,Y 263.363,Z 407.677,A -85,B 0,C 180,E1 -18280.76,E2 -18280.76} C_VEL
LIN {X 0,Y 263.337,Z 407.68,A -85,B 0,C 180,E1 -18285.472,E2 -18285.472} C_VEL
LIN {X 0,Y 263.247,Z 407.694,A -85,B 0,C 180,E1 -18290.301,E2 -18290.301} C_VEL
LIN {X 0,Y 263.1,Z 407.71,A -85,B 0,C 180,E1 -18294.744,E2 -18294.744} C_VEL
LIN {X 0,Y 262.893,Z 407.739,A -85,B 0,C 180,E1 -18298.095,E2 -18298.095} C_VEL
LIN {X 0,Y 262.52,Z 407.782,A -85,B 0,C 180,E1 -18301.057,E2 -18301.057} C_VEL
LIN {X 0,Y 262.081,Z 407.847,A -85,B 0,C 180,E1 -18304.265,E2 -18304.265} C_VEL
LIN {X 0,Y 261.935,Z 409.531,A -85,B 0,C 180,E1 -18307.094,E2 -18307.094} C_VEL
LIN {X 0,Y 261.945,Z 409.8,A -85,B 0,C 180,E1 -18307.436,E2 -18307.436} C_VEL
LIN {X 0,Y 265.003,Z 422.626,A -85,B 0,C 180,E1 -18308.425,E2 -18308.425} C_VEL
LIN {X 0,Y 267.905,Z 436.011,A -85,B 0,C 180,E1 -18309.742,E2 -18309.742} C_VEL
LIN {X 0,Y 269.695,Z 445.88,A -85,B 0,C 180,E1 -18310.915,E2 -18310.915} C_VEL
LIN {X 0,Y 268.405,Z 456.83,A -85,B 0,C 180,E1 -18312.296,E2 -18312.296} C_VEL
LIN {X 0,Y 266.868,Z 468.432,A -85,B 0,C 180,E1 -18314.143,E2 -18314.143} C_VEL
LIN {X 0,Y 265.438,Z 478.906,A -85,B 0,C 180,E1 -18316.23,E2 -18316.23} C_VEL
LIN {X 0,Y 264.162,Z 487.314,A -85,B 0,C 180,E1 -18318.31,E2 -18318.31} C_VEL
LIN {X 0,Y 263.105,Z 495.302,A -85,B 0,C 180,E1 -18320.761,E2 -18320.761} C_VEL
LIN {X 0,Y 262.391,Z 500.694,A -85,B 0,C 180,E1 -18322.823,E2 -18322.823} C_VEL
LIN {X 0,Y 261.781,Z 506.517,A -85,B 0,C 180,E1 -18325.684,E2 -18325.684} C_VEL
LIN {X 0,Y 261.331,Z 510.463,A -85,B 0,C 180,E1 -18328.373,E2 -18328.373} C_VEL
LIN {X 0,Y 261.113,Z 513.057,A -85,B 0,C 180,E1 -18331.023,E2 -18331.023} C_VEL
LIN {X 0,Y 261.145,Z 514.091,A -85,B 0,C 180,E1 -18332.775,E2 -18332.775} C_VEL
LIN {X 0,Y 261.29,Z 514.607,A -85,B 0,C 180,E1 -18334.511,E2 -18334.511} C_VEL
LIN {X 0,Y 261.592,Z 514.647,A -85,B 0,C 180,E1 -18336.236,E2 -18336.236} C_VEL
LIN {X 0,Y 262.015,Z 514.147,A -85,B 0,C 180,E1 -18337.945,E2 -18337.945} C_VEL
LIN {X 0,Y 262.606,Z 513.197,A -85,B 0,C 180,E1 -18339.642,E2 -18339.642} C_VEL
LIN {X 0,Y 263.278,Z 511.759,A -85,B 0,C 180,E1 -18341.319,E2 -18341.319} C_VEL
LIN {X 0,Y 264.619,Z 508.507,A -85,B 0,C 180,E1 -18343.931,E2 -18343.931} C_VEL
LIN {X 0,Y 266.176,Z 504.484,A -85,B 0,C 180,E1 -18346.255,E2 -18346.255} C_VEL
LIN {X 0,Y 268.284,Z 498.962,A -85,B 0,C 180,E1 -18348.671,E2 -18348.671} C_VEL
LIN {X 0,Y 270.707,Z 492.027,A -85,B 0,C 180,E1 -18351.04,E2 -18351.04} C_VEL
LIN {X 0,Y 273.586,Z 483.286,A -85,B 0,C 180,E1 -18353.363,E2 -18353.363} C_VEL
LIN {X 0,Y 276.481,Z 473.766,A -85,B 0,C 180,E1 -18355.377,E2 -18355.377} C_VEL
LIN {X 0,Y 279.251,Z 463.381,A -85,B 0,C 180,E1 -18357.116,E2 -18357.116} C_VEL
LIN {X 0,Y 280.098,Z 459.667,A -85,B 0,C 180,E1 -18357.665,E2 -18357.665} C_VEL
LIN {X 0,Y 278.592,Z 450.111,A -85,B 0,C 180,E1 -18359.512,E2 -18359.512} C_VEL
LIN {X 0,Y 274.657,Z 437.115,A -85,B 0,C 180,E1 -18362.08,E2 -18362.08} C_VEL
LIN {X 0,Y 272.119,Z 430.735,A -85,B 0,C 180,E1 -18363.382,E2 -18363.382} C_VEL
LIN {X 0,Y 268.765,Z 424.469,A -85,B 0,C 180,E1 -18364.81,E2 -18364.81} C_VEL
LIN {X 0,Y 266.807,Z 420.714,A -85,B 0,C 180,E1 -18365.67,E2 -18365.67} C_VEL
LIN {X 0,Y 264.932,Z 417.826,A -85,B 0,C 180,E1 -18366.427,E2 -18366.427} C_VEL
LIN {X 0,Y 264.498,Z 416.263,A -85,B 0,C 180,E1 -18366.677,E2 -18366.677} C_VEL
LIN {X 0,Y 264.563,Z 415.052,A -85,B 0,C 180,E1 -18370.654,E2 -18370.654} C_VEL
LIN {X 0,Y 264.366,Z 414.101,A -85,B 0,C 180,E1 -18375.418,E2 -18375.418} C_VEL
LIN {X 0,Y 264.292,Z 413.857,A -85,B 0,C 180,E1 -18377.444,E2 -18377.444} C_VEL
LIN {X 0,Y 263.6,Z 413.914,A -85,B 0,C 180,E1 -18378.717,E2 -18378.717} C_VEL
LIN {X 0,Y 260.81,Z 414.482,A -85,B 0,C 180,E1 -18380.792,E2 -18380.792} C_VEL
LIN {X 0,Y 258.464,Z 415.052,A -85,B 0,C 180,E1 -18382.479,E2 -18382.479} C_VEL
LIN {X 0,Y 257.455,Z 415.377,A -85,B 0,C 180,E1 -18383.786,E2 -18383.786} C_VEL
LIN {X 0,Y 257.371,Z 415.429,A -85,B 0,C 180,E1 -18384.229,E2 -18384.229} C_VEL
LIN {X 0,Y 257.431,Z 415.9,A -85,B 0,C 180,E1 -18387.654,E2 -18387.654} C_VEL
LIN {X 0,Y 257.544,Z 416.789,A -85,B 0,C 180,E1 -18391.232,E2 -18391.232} C_VEL
LIN {X 0,Y 257.803,Z 418.17,A -85,B 0,C 180,E1 -18395.144,E2 -18395.144} C_VEL
LIN {X 0,Y 258.099,Z 419.885,A -85,B 0,C 180,E1 -18398.778,E2 -18398.778} C_VEL
LIN {X 0,Y 258.563,Z 422.296,A -85,B 0,C 180,E1 -18402.808,E2 -18402.808} C_VEL
LIN {X 0,Y 258.819,Z 423.892,A -85,B 0,C 180,E1 -18405.099,E2 -18405.099} C_VEL
LIN {X 0,Y 259.1,Z 425.596,A -85,B 0,C 180,E1 -18407.313,E2 -18407.313} C_VEL
LIN {X 0,Y 259.316,Z 427.408,A -85,B 0,C 180,E1 -18409.434,E2 -18409.434} C_VEL
LIN {X 0,Y 259.482,Z 429.545,A -85,B 0,C 180,E1 -18411.765,E2 -18411.765} C_VEL
LIN {X 0,Y 259.26,Z 431.717,A -85,B 0,C 180,E1 -18413.839,E2 -18413.839} C_VEL
LIN {X 0,Y 260.424,Z 435.518,A -85,B 0,C 180,E1 -18414.47,E2 -18414.47} C_VEL
LIN {X 0,Y 261.431,Z 437.657,A -85,B 0,C 180,E1 -18414.932,E2 -18414.932} C_VEL
LIN {X 0,Y 264.419,Z 446.846,A -85,B 0,C 180,E1 -18416.595,E2 -18416.595} C_VEL
LIN {X 0,Y 267.447,Z 458.831,A -85,B 0,C 180,E1 -18418.654,E2 -18418.654} C_VEL
LIN {X 0,Y 269.18,Z 471.089,A -85,B 0,C 180,E1 -18420.698,E2 -18420.698} C_VEL
LIN {X 0,Y 269.542,Z 481.404,A -85,B 0,C 180,E1 -18422.44,E2 -18422.44} C_VEL
LIN {X 0,Y 268.9,Z 491.533,A -85,B 0,C 180,E1 -18424.253,E2 -18424.253} C_VEL
LIN {X 0,Y 268.13,Z 496.631,A -85,B 0,C 180,E1 -18425.212,E2 -18425.212} C_VEL
LIN {X 0,Y 265.305,Z 505.752,A -85,B 0,C 180,E1 -18427.007,E2 -18427.007} C_VEL
LIN {X 0,Y 262.238,Z 514.765,A -85,B 0,C 180,E1 -18429.207,E2 -18429.207} C_VEL
LIN {X 0,Y 259.446,Z 523.304,A -85,B 0,C 180,E1 -18431.856,E2 -18431.856} C_VEL
LIN {X 0,Y 257.678,Z 529.197,A -85,B 0,C 180,E1 -18434.179,E2 -18434.179} C_VEL
LIN {X 0,Y 256.044,Z 533.94,A -85,B 0,C 180,E1 -18436.514,E2 -18436.514} C_VEL
LIN {X 0,Y 255.025,Z 537.633,A -85,B 0,C 180,E1 -18438.884,E2 -18438.884} C_VEL
LIN {X 0,Y 254.29,Z 541.069,A -85,B 0,C 180,E1 -18442.063,E2 -18442.063} C_VEL
LIN {X 0,Y 254.087,Z 542.72,A -85,B 0,C 180,E1 -18444.729,E2 -18444.729} C_VEL
LIN {X 0,Y 254.182,Z 543.256,A -85,B 0,C 180,E1 -18446.836,E2 -18446.836} C_VEL
LIN {X 0,Y 254.385,Z 542.648,A -85,B 0,C 180,E1 -18450.006,E2 -18450.006} C_VEL
LIN {X 0,Y 254.277,Z 541.722,A -85,B 0,C 180,E1 -18451.59,E2 -18451.59} C_VEL
LIN {X 0,Y 254.261,Z 540.361,A -85,B 0,C 180,E1 -18453.175,E2 -18453.175} C_VEL
LIN {X 0,Y 254.309,Z 537.102,A -85,B 0,C 180,E1 -18455.787,E2 -18455.787} C_VEL
LIN {X 0,Y 254.529,Z 531.821,A -85,B 0,C 180,E1 -18458.741,E2 -18458.741} C_VEL
LIN {X 0,Y 254.963,Z 526.174,A -85,B 0,C 180,E1 -18461.131,E2 -18461.131} C_VEL
LIN {X 0,Y 255.853,Z 519.082,A -85,B 0,C 180,E1 -18463.508,E2 -18463.508} C_VEL
LIN {X 0,Y 257.057,Z 510.246,A -85,B 0,C 180,E1 -18465.872,E2 -18465.872} C_VEL
LIN {X 0,Y 258.109,Z 502.207,A -85,B 0,C 180,E1 -18467.631,E2 -18467.631} C_VEL
LIN {X 0,Y 259.566,Z 492.543,A -85,B 0,C 180,E1 -18469.376,E2 -18469.376} C_VEL
LIN {X 0,Y 260.319,Z 486.196,A -85,B 0,C 180,E1 -18470.346,E2 -18470.346} C_VEL
LIN {X 0,Y 259.658,Z 475.116,A -85,B 0,C 180,E1 -18471.854,E2 -18471.854} C_VEL
LIN {X 0,Y 258.511,Z 462.686,A -85,B 0,C 180,E1 -18473.244,E2 -18473.244} C_VEL
LIN {X 0,Y 257.017,Z 449.261,A -85,B 0,C 180,E1 -18474.409,E2 -18474.409} C_VEL
LIN {X 0,Y 255.588,Z 437.872,A -85,B 0,C 180,E1 -18475.198,E2 -18475.198} C_VEL
LIN {X 0,Y 256.511,Z 431.969,A -85,B 0,C 180,E1 -18479.555,E2 -18479.555} C_VEL
LIN {X 0,Y 257.706,Z 426.036,A -85,B 0,C 180,E1 -18483.997,E2 -18483.997} C_VEL
LIN {X 0,Y 258.345,Z 422.401,A -85,B 0,C 180,E1 -18486.767,E2 -18486.767} C_VEL
LIN {X 0,Y 258.197,Z 419.907,A -85,B 0,C 180,E1 -18488.765,E2 -18488.765} C_VEL
LIN {X 0,Y 257.268,Z 414.774,A -85,B 0,C 180,E1 -18493.08,E2 -18493.08} C_VEL
LIN {X 0,Y 256.488,Z 410.61,A -85,B 0,C 180,E1 -18496.761,E2 -18496.761} C_VEL
LIN {X 0,Y 256.08,Z 408.589,A -85,B 0,C 180,E1 -18498.8,E2 -18498.8} C_VEL
LIN {X 0,Y 256.136,Z 408.579,A -85,B 0,C 180,E1 -18502.867,E2 -18502.867} C_VEL
LIN {X 0,Y 256.084,Z 408.584,A -85,B 0,C 180,E1 -18506.708,E2 -18506.708} C_VEL
LIN {X 0,Y 256.073,Z 408.585,A -85,B 0,C 180,E1 -18510.394,E2 -18510.394} C_VEL
LIN {X 0,Y 256.151,Z 408.577,A -85,B 0,C 180,E1 -18514.889,E2 -18514.889} C_VEL
LIN {X 0,Y 256.142,Z 408.58,A -85,B 0,C 180,E1 -18519.101,E2 -18519.101} C_VEL
LIN {X 0,Y 256.249,Z 408.563,A -85,B 0,C 180,E1 -18524.08,E2 -18524.08} C_VEL
LIN {X 0,Y 256.305,Z 408.559,A -85,B 0,C 180,E1 -18528.932,E2 -18528.932} C_VEL
LIN {X 0,Y 256.515,Z 408.529,A -85,B 0,C 180,E1 -18532.125,E2 -18532.125} C_VEL
LIN {X 0,Y 256.507,Z 408.535,A -85,B 0,C 180,E1 -18536.857,E2 -18536.857} C_VEL
LIN {X 0,Y 256.759,Z 408.499,A -85,B 0,C 180,E1 -18539.999,E2 -18539.999} C_VEL
LIN {X 0,Y 256.473,Z 408.538,A -85,B 0,C 180,E1 -18543.14,E2 -18543.14} C_VEL
LIN {X 0,Y 256.484,Z 408.533,A -85,B 0,C 180,E1 -18547.873,E2 -18547.873} C_VEL
LIN {X 0,Y 256.302,Z 408.559,A -85,B 0,C 180,E1 -18551.065,E2 -18551.065} C_VEL
LIN {X 0,Y 256.245,Z 408.562,A -85,B 0,C 180,E1 -18555.917,E2 -18555.917} C_VEL
LIN {X 0,Y 256.139,Z 408.579,A -85,B 0,C 180,E1 -18560.896,E2 -18560.896} C_VEL
LIN {X 0,Y 256.183,Z 408.572,A -85,B 0,C 180,E1 -18565.126,E2 -18565.126} C_VEL
LIN {X 0,Y 256.127,Z 408.582,A -85,B 0,C 180,E1 -18568.582,E2 -18568.582} C_VEL
LIN {X 0,Y 256.086,Z 408.581,A -85,B 0,C 180,E1 -18571.697,E2 -18571.697} C_VEL
LIN {X 0,Y 256.092,Z 408.583,A -85,B 0,C 180,E1 -18575.189,E2 -18575.189} C_VEL
LIN {X 0,Y 256.123,Z 408.579,A -85,B 0,C 180,E1 -18577.266,E2 -18577.266} C_VEL
LIN {X 0,Y 256.064,Z 408.586,A -85,B 0,C 180,E1 -18581.199,E2 -18581.199} C_VEL
LIN {X 0,Y 256.049,Z 408.588,A -85,B 0,C 180,E1 -18585.53,E2 -18585.53} C_VEL
LIN {X 0,Y 256.058,Z 408.588,A -85,B 0,C 180,E1 -18588.791,E2 -18588.791} C_VEL
LIN {X 0,Y 256.136,Z 408.579,A -85,B 0,C 180,E1 -18592.863,E2 -18592.863} C_VEL
LIN {X 0,Y 256.073,Z 408.586,A -85,B 0,C 180,E1 -18596.702,E2 -18596.702} C_VEL
LIN {X 0,Y 256.115,Z 408.584,A -85,B 0,C 180,E1 -18600.395,E2 -18600.395} C_VEL
LIN {X 0,Y 256.191,Z 408.569,A -85,B 0,C 180,E1 -18604.856,E2 -18604.856} C_VEL
LIN {X 0,Y 256.171,Z 408.573,A -85,B 0,C 180,E1 -18609.1,E2 -18609.1} C_VEL
LIN {X 0,Y 256.3,Z 408.558,A -85,B 0,C 180,E1 -18614.08,E2 -18614.08} C_VEL
LIN {X 0,Y 256.295,Z 408.558,A -85,B 0,C 180,E1 -18618.928,E2 -18618.928} C_VEL
LIN {X 0,Y 256.512,Z 408.532,A -85,B 0,C 180,E1 -18622.121,E2 -18622.121} C_VEL
LIN {X 0,Y 256.492,Z 408.533,A -85,B 0,C 180,E1 -18626.853,E2 -18626.853} C_VEL
LIN {X 0,Y 256.758,Z 408.502,A -85,B 0,C 180,E1 -18629.994,E2 -18629.994} C_VEL
LIN {X 0,Y 256.492,Z 408.533,A -85,B 0,C 180,E1 -18633.136,E2 -18633.136} C_VEL
LIN {X 0,Y 256.53,Z 408.53,A -85,B 0,C 180,E1 -18637.867,E2 -18637.867} C_VEL
LIN {X 0,Y 256.298,Z 408.557,A -85,B 0,C 180,E1 -18641.06,E2 -18641.06} C_VEL
LIN {X 0,Y 256.286,Z 408.561,A -85,B 0,C 180,E1 -18645.909,E2 -18645.909} C_VEL
LIN {X 0,Y 256.147,Z 408.576,A -85,B 0,C 180,E1 -18650.89,E2 -18650.89} C_VEL
LIN {X 0,Y 256.049,Z 408.588,A -85,B 0,C 180,E1 -18655.076,E2 -18655.076} C_VEL
LIN {X 0,Y 255.794,Z 408.621,A -85,B 0,C 180,E1 -18658.457,E2 -18658.457} C_VEL
LIN {X 0,Y 255.407,Z 408.67,A -85,B 0,C 180,E1 -18661.514,E2 -18661.514} C_VEL
LIN {X 0,Y 254.907,Z 408.953,A -85,B 0,C 180,E1 -18665.371,E2 -18665.371} C_VEL
LIN {X 0,Y 254.884,Z 410.171,A -85,B 0,C 180,E1 -18666.967,E2 -18666.967} C_VEL
LIN {X 0,Y 258.477,Z 425.318,A -85,B 0,C 180,E1 -18668.203,E2 -18668.203} C_VEL
LIN {X 0,Y 261.107,Z 437.577,A -85,B 0,C 180,E1 -18669.477,E2 -18669.477} C_VEL
LIN {X 0,Y 262.725,Z 446.629,A -85,B 0,C 180,E1 -18670.603,E2 -18670.603} C_VEL
LIN {X 0,Y 261.596,Z 456.321,A -85,B 0,C 180,E1 -18671.855,E2 -18671.855} C_VEL
LIN {X 0,Y 260.066,Z 467.583,A -85,B 0,C 180,E1 -18673.651,E2 -18673.651} C_VEL
LIN {X 0,Y 258.523,Z 478.559,A -85,B 0,C 180,E1 -18675.846,E2 -18675.846} C_VEL
LIN {X 0,Y 257.194,Z 487.078,A -85,B 0,C 180,E1 -18677.975,E2 -18677.975} C_VEL
LIN {X 0,Y 256.224,Z 494.21,A -85,B 0,C 180,E1 -18680.165,E2 -18680.165} C_VEL
LIN {X 0,Y 255.322,Z 500.932,A -85,B 0,C 180,E1 -18682.732,E2 -18682.732} C_VEL
LIN {X 0,Y 254.759,Z 506.201,A -85,B 0,C 180,E1 -18685.313,E2 -18685.313} C_VEL
LIN {X 0,Y 254.37,Z 509.465,A -85,B 0,C 180,E1 -18687.402,E2 -18687.402} C_VEL
LIN {X 0,Y 254.049,Z 512.602,A -85,B 0,C 180,E1 -18690.137,E2 -18690.137} C_VEL
LIN {X 0,Y 254.057,Z 514.135,A -85,B 0,C 180,E1 -18692.262,E2 -18692.262} C_VEL
LIN {X 0,Y 254.108,Z 514.8,A -85,B 0,C 180,E1 -18693.737,E2 -18693.737} C_VEL
LIN {X 0,Y 254.413,Z 515.124,A -85,B 0,C 180,E1 -18695.71,E2 -18695.71} C_VEL
LIN {X 0,Y 254.736,Z 514.948,A -85,B 0,C 180,E1 -18697.28,E2 -18697.28} C_VEL
LIN {X 0,Y 255.389,Z 514.155,A -85,B 0,C 180,E1 -18699.31,E2 -18699.31} C_VEL
LIN {X 0,Y 256.723,Z 511.572,A -85,B 0,C 180,E1 -18702.476,E2 -18702.476} C_VEL
LIN {X 0,Y 258.243,Z 508.242,A -85,B 0,C 180,E1 -18705.018,E2 -18705.018} C_VEL
LIN {X 0,Y 260.138,Z 503.726,A -85,B 0,C 180,E1 -18707.52,E2 -18707.52} C_VEL
LIN {X 0,Y 262.874,Z 496.768,A -85,B 0,C 180,E1 -18710.382,E2 -18710.382} C_VEL
LIN {X 0,Y 265.709,Z 489.177,A -85,B 0,C 180,E1 -18712.784,E2 -18712.784} C_VEL
LIN {X 0,Y 268.56,Z 480.54,A -85,B 0,C 180,E1 -18714.937,E2 -18714.937} C_VEL
LIN {X 0,Y 271.61,Z 470.832,A -85,B 0,C 180,E1 -18716.849,E2 -18716.849} C_VEL
LIN {X 0,Y 273.805,Z 462.81,A -85,B 0,C 180,E1 -18718.163,E2 -18718.163} C_VEL
LIN {X 0,Y 273.737,Z 459.039,A -85,B 0,C 180,E1 -18718.898,E2 -18718.898} C_VEL
LIN {X 0,Y 272.589,Z 452.231,A -85,B 0,C 180,E1 -18720.318,E2 -18720.318} C_VEL
LIN {X 0,Y 268.955,Z 439.567,A -85,B 0,C 180,E1 -18722.997,E2 -18722.997} C_VEL
LIN {X 0,Y 266.794,Z 434.05,A -85,B 0,C 180,E1 -18724.215,E2 -18724.215} C_VEL
LIN {X 0,Y 262.881,Z 426.252,A -85,B 0,C 180,E1 -18726.14,E2 -18726.14} C_VEL
LIN {X 0,Y 260.812,Z 422.809,A -85,B 0,C 180,E1 -18727.076,E2 -18727.076} C_VEL
LIN {X 0,Y 260.158,Z 421.602,A -85,B 0,C 180,E1 -18727.388,E2 -18727.388} C_VEL
LIN {X 0,Y 258.146,Z 418.768,A -85,B 0,C 180,E1 -18728.293,E2 -18728.293} C_VEL
LIN {X 0,Y 257.621,Z 417.073,A -85,B 0,C 180,E1 -18728.631,E2 -18728.631} C_VEL
LIN {X 0,Y 257.584,Z 416.466,A -85,B 0,C 180,E1 -18731.012,E2 -18731.012} C_VEL
LIN {X 0,Y 257.424,Z 415.586,A -85,B 0,C 180,E1 -18735.845,E2 -18735.845} C_VEL
LIN {X 0,Y 257.345,Z 415.315,A -85,B 0,C 180,E1 -18739.132,E2 -18739.132} C_VEL
LIN {X 0,Y 257.335,Z 415.319,A -85,B 0,C 180,E1 -18742.481,E2 -18742.481} C_VEL
LIN {X 0,Y 257.371,Z 415.429,A -85,B 0,C 180,E1 -18744.229,E2 -18744.229} C_VEL
LIN {X 0,Y 256.712,Z 415.746,A -85,B 0,C 180,E1 -18745.535,E2 -18745.535} C_VEL
LIN {X 0,Y 253.944,Z 416.758,A -85,B 0,C 180,E1 -18747.66,E2 -18747.66} C_VEL
LIN {X 0,Y 251.627,Z 417.701,A -85,B 0,C 180,E1 -18749.388,E2 -18749.388} C_VEL
LIN {X 0,Y 250.676,Z 418.285,A -85,B 0,C 180,E1 -18750.727,E2 -18750.727} C_VEL
LIN {X 0,Y 250.62,Z 418.435,A -85,B 0,C 180,E1 -18751.181,E2 -18751.181} C_VEL
LIN {X 0,Y 250.786,Z 419.411,A -85,B 0,C 180,E1 -18754.09,E2 -18754.09} C_VEL
LIN {X 0,Y 251.152,Z 421.328,A -85,B 0,C 180,E1 -18758.427,E2 -18758.427} C_VEL
LIN {X 0,Y 251.547,Z 423.405,A -85,B 0,C 180,E1 -18762.11,E2 -18762.11} C_VEL
LIN {X 0,Y 252.039,Z 426.441,A -85,B 0,C 180,E1 -18766.47,E2 -18766.47} C_VEL
LIN {X 0,Y 252.368,Z 429.477,A -85,B 0,C 180,E1 -18770.179,E2 -18770.179} C_VEL
LIN {X 0,Y 252.547,Z 431.03,A -85,B 0,C 180,E1 -18771.723,E2 -18771.723} C_VEL
LIN {X 0,Y 253.56,Z 434.277,A -85,B 0,C 180,E1 -18772.345,E2 -18772.345} C_VEL
LIN {X 0,Y 255.286,Z 437.345,A -85,B 0,C 180,E1 -18773.19,E2 -18773.19} C_VEL
LIN {X 0,Y 258.281,Z 446.202,A -85,B 0,C 180,E1 -18774.994,E2 -18774.994} C_VEL
LIN {X 0,Y 261.212,Z 458.066,A -85,B 0,C 180,E1 -18777.226,E2 -18777.226} C_VEL
LIN {X 0,Y 262.753,Z 467.17,A -85,B 0,C 180,E1 -18778.864,E2 -18778.864} C_VEL
LIN {X 0,Y 263.487,Z 477.237,A -85,B 0,C 180,E1 -18780.674,E2 -18780.674} C_VEL
LIN {X 0,Y 263.212,Z 488.021,A -85,B 0,C 180,E1 -18782.649,E2 -18782.649} C_VEL
LIN {X 0,Y 261.78,Z 497.76,A -85,B 0,C 180,E1 -18784.568,E2 -18784.568} C_VEL
LIN {X 0,Y 258.315,Z 508.142,A -85,B 0,C 180,E1 -18786.772,E2 -18786.772} C_VEL
LIN {X 0,Y 255.175,Z 516.688,A -85,B 0,C 180,E1 -18789.027,E2 -18789.027} C_VEL
LIN {X 0,Y 252.511,Z 524.216,A -85,B 0,C 180,E1 -18791.574,E2 -18791.574} C_VEL
LIN {X 0,Y 250.844,Z 529.336,A -85,B 0,C 180,E1 -18793.736,E2 -18793.736} C_VEL
LIN {X 0,Y 249.12,Z 533.946,A -85,B 0,C 180,E1 -18796.132,E2 -18796.132} C_VEL
LIN {X 0,Y 248.037,Z 537.539,A -85,B 0,C 180,E1 -18798.566,E2 -18798.566} C_VEL
LIN {X 0,Y 247.219,Z 540.829,A -85,B 0,C 180,E1 -18801.835,E2 -18801.835} C_VEL
LIN {X 0,Y 246.987,Z 542.471,A -85,B 0,C 180,E1 -18804.836,E2 -18804.836} C_VEL
LIN {X 0,Y 247.108,Z 542.804,A -85,B 0,C 180,E1 -18806.745,E2 -18806.745} C_VEL
LIN {X 0,Y 247.302,Z 542.096,A -85,B 0,C 180,E1 -18810.006,E2 -18810.006} C_VEL
LIN {X 0,Y 247.198,Z 541.107,A -85,B 0,C 180,E1 -18811.635,E2 -18811.635} C_VEL
LIN {X 0,Y 247.195,Z 539.65,A -85,B 0,C 180,E1 -18813.266,E2 -18813.266} C_VEL
LIN {X 0,Y 247.233,Z 536.566,A -85,B 0,C 180,E1 -18815.76,E2 -18815.76} C_VEL
LIN {X 0,Y 247.366,Z 532.499,A -85,B 0,C 180,E1 -18818.173,E2 -18818.173} C_VEL
LIN {X 0,Y 247.875,Z 526.142,A -85,B 0,C 180,E1 -18821.039,E2 -18821.039} C_VEL
LIN {X 0,Y 248.72,Z 519.188,A -85,B 0,C 180,E1 -18823.486,E2 -18823.486} C_VEL
LIN {X 0,Y 249.92,Z 510.477,A -85,B 0,C 180,E1 -18825.919,E2 -18825.919} C_VEL
LIN {X 0,Y 250.9,Z 503.024,A -85,B 0,C 180,E1 -18827.635,E2 -18827.635} C_VEL
LIN {X 0,Y 252.477,Z 493.093,A -85,B 0,C 180,E1 -18829.519,E2 -18829.519} C_VEL
LIN {X 0,Y 253.31,Z 486.953,A -85,B 0,C 180,E1 -18830.51,E2 -18830.51} C_VEL
LIN {X 0,Y 252.693,Z 476.109,A -85,B 0,C 180,E1 -18832.059,E2 -18832.059} C_VEL
LIN {X 0,Y 251.547,Z 463.079,A -85,B 0,C 180,E1 -18833.575,E2 -18833.575} C_VEL
LIN {X 0,Y 250.098,Z 449.978,A -85,B 0,C 180,E1 -18834.769,E2 -18834.769} C_VEL
LIN {X 0,Y 248.576,Z 437.568,A -85,B 0,C 180,E1 -18835.634,E2 -18835.634} C_VEL
LIN {X 0,Y 249.644,Z 431.249,A -85,B 0,C 180,E1 -18840.452,E2 -18840.452} C_VEL
LIN {X 0,Y 250.867,Z 425.479,A -85,B 0,C 180,E1 -18844.922,E2 -18844.922} C_VEL
LIN {X 0,Y 251.279,Z 422.891,A -85,B 0,C 180,E1 -18846.971,E2 -18846.971} C_VEL
LIN {X 0,Y 250.882,Z 419.116,A -85,B 0,C 180,E1 -18850.12,E2 -18850.12} C_VEL
LIN {X 0,Y 249.885,Z 413.928,A -85,B 0,C 180,E1 -18854.685,E2 -18854.685} C_VEL
LIN {X 0,Y 249.054,Z 409.465,A -85,B 0,C 180,E1 -18858.862,E2 -18858.862} C_VEL
LIN {X 0,Y 249.053,Z 409.459,A -85,B 0,C 180,E1 -18862.205,E2 -18862.205} C_VEL
LIN {X 0,Y 249.061,Z 409.458,A -85,B 0,C 180,E1 -18865.641,E2 -18865.641} C_VEL
LIN {X 0,Y 249.02,Z 409.466,A -85,B 0,C 180,E1 -18869.467,E2 -18869.467} C_VEL
LIN {X 0,Y 249.053,Z 409.461,A -85,B 0,C 180,E1 -18873.159,E2 -18873.159} C_VEL
LIN {X 0,Y 249.07,Z 409.459,A -85,B 0,C 180,E1 -18876.73,E2 -18876.73} C_VEL
LIN {X 0,Y 249.076,Z 409.456,A -85,B 0,C 180,E1 -18880.207,E2 -18880.207} C_VEL
LIN {X 0,Y 249.177,Z 409.444,A -85,B 0,C 180,E1 -18883.616,E2 -18883.616} C_VEL
LIN {X 0,Y 249.248,Z 409.436,A -85,B 0,C 180,E1 -18888.615,E2 -18888.615} C_VEL
LIN {X 0,Y 249.455,Z 409.409,A -85,B 0,C 180,E1 -18891.901,E2 -18891.901} C_VEL
LIN {X 0,Y 249.299,Z 409.431,A -85,B 0,C 180,E1 -18895.147,E2 -18895.147} C_VEL
LIN {X 0,Y 249.689,Z 409.379,A -85,B 0,C 180,E1 -18898.386,E2 -18898.386} C_VEL
LIN {X 0,Y 249.679,Z 409.382,A -85,B 0,C 180,E1 -18901.612,E2 -18901.612} C_VEL
LIN {X 0,Y 249.434,Z 409.411,A -85,B 0,C 180,E1 -18906.604,E2 -18906.604} C_VEL
LIN {X 0,Y 249.35,Z 409.422,A -85,B 0,C 180,E1 -18909.735,E2 -18909.735} C_VEL
LIN {X 0,Y 249.186,Z 409.445,A -85,B 0,C 180,E1 -18914.703,E2 -18914.703} C_VEL
LIN {X 0,Y 249.109,Z 409.453,A -85,B 0,C 180,E1 -18918.078,E2 -18918.078} C_VEL
LIN {X 0,Y 249.061,Z 409.458,A -85,B 0,C 180,E1 -18921.519,E2 -18921.519} C_VEL
LIN {X 0,Y 249.13,Z 409.45,A -85,B 0,C 180,E1 -18925.471,E2 -18925.471} C_VEL
LIN {X 0,Y 249.068,Z 409.459,A -85,B 0,C 180,E1 -18928.978,E2 -18928.978} C_VEL
LIN {X 0,Y 249.039,Z 409.462,A -85,B 0,C 180,E1 -18932.423,E2 -18932.423} C_VEL
LIN {X 0,Y 249.058,Z 409.462,A -85,B 0,C 180,E1 -18936.339,E2 -18936.339} C_VEL
LIN {X 0,Y 249.016,Z 409.466,A -85,B 0,C 180,E1 -18940.474,E2 -18940.474} C_VEL
LIN {X 0,Y 248.994,Z 409.469,A -85,B 0,C 180,E1 -18944.879,E2 -18944.879} C_VEL
LIN {X 0,Y 249.014,Z 409.463,A -85,B 0,C 180,E1 -18947.356,E2 -18947.356} C_VEL
LIN {X 0,Y 249.05,Z 409.462,A -85,B 0,C 180,E1 -18952.196,E2 -18952.196} C_VEL
LIN {X 0,Y 249.05,Z 409.459,A -85,B 0,C 180,E1 -18955.634,E2 -18955.634} C_VEL
LIN {X 0,Y 249.055,Z 409.459,A -85,B 0,C 180,E1 -18959.468,E2 -18959.468} C_VEL
LIN {X 0,Y 249.076,Z 409.456,A -85,B 0,C 180,E1 -18963.157,E2 -18963.157} C_VEL
LIN {X 0,Y 249.084,Z 409.457,A -85,B 0,C 180,E1 -18966.727,E2 -18966.727} C_VEL
LIN {X 0,Y 249.113,Z 409.456,A -85,B 0,C 180,E1 -18970.206,E2 -18970.206} C_VEL
LIN {X 0,Y 249.242,Z 409.434,A -85,B 0,C 180,E1 -18973.616,E2 -18973.616} C_VEL
LIN {X 0,Y 249.243,Z 409.438,A -85,B 0,C 180,E1 -18978.61,E2 -18978.61} C_VEL
LIN {X 0,Y 249.451,Z 409.41,A -85,B 0,C 180,E1 -18981.896,E2 -18981.896} C_VEL
LIN {X 0,Y 249.29,Z 409.43,A -85,B 0,C 180,E1 -18985.143,E2 -18985.143} C_VEL
LIN {X 0,Y 249.669,Z 409.384,A -85,B 0,C 180,E1 -18988.381,E2 -18988.381} C_VEL
LIN {X 0,Y 249.669,Z 409.382,A -85,B 0,C 180,E1 -18991.607,E2 -18991.607} C_VEL
LIN {X 0,Y 249.452,Z 409.411,A -85,B 0,C 180,E1 -18996.465,E2 -18996.465} C_VEL
LIN {X 0,Y 249.413,Z 409.414,A -85,B 0,C 180,E1 -18999.727,E2 -18999.727} C_VEL
LIN {X 0,Y 249.193,Z 409.442,A -85,B 0,C 180,E1 -19004.698,E2 -19004.698} C_VEL
LIN {X 0,Y 249.124,Z 409.453,A -85,B 0,C 180,E1 -19008.072,E2 -19008.072} C_VEL
LIN {X 0,Y 249.066,Z 409.459,A -85,B 0,C 180,E1 -19011.513,E2 -19011.513} C_VEL
LIN {X 0,Y 248.961,Z 409.472,A -85,B 0,C 180,E1 -19015.404,E2 -19015.404} C_VEL
LIN {X 0,Y 248.689,Z 409.505,A -85,B 0,C 180,E1 -19018.832,E2 -19018.832} C_VEL
LIN {X 0,Y 248.188,Z 409.571,A -85,B 0,C 180,E1 -19022.541,E2 -19022.541} C_VEL
LIN {X 0,Y 247.85,Z 409.856,A -85,B 0,C 180,E1 -19025.559,E2 -19025.559} C_VEL
LIN {X 0,Y 247.809,Z 410.563,A -85,B 0,C 180,E1 -19026.483,E2 -19026.483} C_VEL
LIN {X 0,Y 251.469,Z 425.872,A -85,B 0,C 180,E1 -19027.793,E2 -19027.793} C_VEL
LIN {X 0,Y 253.992,Z 437.694,A -85,B 0,C 180,E1 -19029.056,E2 -19029.056} C_VEL
LIN {X 0,Y 255.763,Z 448.387,A -85,B 0,C 180,E1 -19030.42,E2 -19030.42} C_VEL
LIN {X 0,Y 254.206,Z 459.857,A -85,B 0,C 180,E1 -19032.014,E2 -19032.014} C_VEL
LIN {X 0,Y 252.829,Z 469.776,A -85,B 0,C 180,E1 -19033.722,E2 -19033.722} C_VEL
LIN {X 0,Y 251.471,Z 479.108,A -85,B 0,C 180,E1 -19035.68,E2 -19035.68} C_VEL
LIN {X 0,Y 250.002,Z 488.439,A -85,B 0,C 180,E1 -19038.116,E2 -19038.116} C_VEL
LIN {X 0,Y 248.973,Z 495.993,A -85,B 0,C 180,E1 -19040.573,E2 -19040.573} C_VEL
LIN {X 0,Y 248.159,Z 501.863,A -85,B 0,C 180,E1 -19042.948,E2 -19042.948} C_VEL
LIN {X 0,Y 247.64,Z 506.692,A -85,B 0,C 180,E1 -19045.419,E2 -19045.419} C_VEL
LIN {X 0,Y 247.134,Z 511.161,A -85,B 0,C 180,E1 -19048.54,E2 -19048.54} C_VEL
LIN {X 0,Y 246.947,Z 514.216,A -85,B 0,C 180,E1 -19051.898,E2 -19051.898} C_VEL
LIN {X 0,Y 247.16,Z 515.422,A -85,B 0,C 180,E1 -19054.755,E2 -19054.755} C_VEL
LIN {X 0,Y 247.49,Z 515.569,A -85,B 0,C 180,E1 -19056.576,E2 -19056.576} C_VEL
LIN {X 0,Y 248.228,Z 514.947,A -85,B 0,C 180,E1 -19059.097,E2 -19059.097} C_VEL
LIN {X 0,Y 249.389,Z 513.109,A -85,B 0,C 180,E1 -19061.943,E2 -19061.943} C_VEL
LIN {X 0,Y 250.842,Z 510.262,A -85,B 0,C 180,E1 -19064.565,E2 -19064.565} C_VEL
LIN {X 0,Y 252.711,Z 506.287,A -85,B 0,C 180,E1 -19067.147,E2 -19067.147} C_VEL
LIN {X 0,Y 255.461,Z 500.02,A -85,B 0,C 180,E1 -19070.101,E2 -19070.101} C_VEL
LIN {X 0,Y 258.248,Z 493.145,A -85,B 0,C 180,E1 -19072.574,E2 -19072.574} C_VEL
LIN {X 0,Y 261.477,Z 484.429,A -85,B 0,C 180,E1 -19075.006,E2 -19075.006} C_VEL
LIN {X 0,Y 264.556,Z 475.637,A -85,B 0,C 180,E1 -19076.956,E2 -19076.956} C_VEL
LIN {X 0,Y 267.483,Z 466.052,A -85,B 0,C 180,E1 -19078.684,E2 -19078.684} C_VEL
LIN {X 0,Y 267.928,Z 462.92,A -85,B 0,C 180,E1 -19079.25,E2 -19079.25} C_VEL
LIN {X 0,Y 267.051,Z 456.25,A -85,B 0,C 180,E1 -19080.722,E2 -19080.722} C_VEL
LIN {X 0,Y 264.171,Z 444.76,A -85,B 0,C 180,E1 -19083.334,E2 -19083.334} C_VEL
LIN {X 0,Y 262.341,Z 439.334,A -85,B 0,C 180,E1 -19084.611,E2 -19084.611} C_VEL
LIN {X 0,Y 258.736,Z 431.628,A -85,B 0,C 180,E1 -19086.63,E2 -19086.63} C_VEL
LIN {X 0,Y 256.426,Z 427.29,A -85,B 0,C 180,E1 -19087.878,E2 -19087.878} C_VEL
LIN {X 0,Y 254.241,Z 423.775,A -85,B 0,C 180,E1 -19088.997,E2 -19088.997} C_VEL
LIN {X 0,Y 253.515,Z 422.667,A -85,B 0,C 180,E1 -19089.355,E2 -19089.355} C_VEL
LIN {X 0,Y 251.399,Z 420.07,A -85,B 0,C 180,E1 -19090.406,E2 -19090.406} C_VEL
LIN {X 0,Y 250.67,Z 417.962,A -85,B 0,C 180,E1 -19090.971,E2 -19090.971} C_VEL
LIN {X 0,Y 250.512,Z 417.325,A -85,B 0,C 180,E1 -19094.626,E2 -19094.626} C_VEL
LIN {X 0,Y 250.434,Z 416.983,A -85,B 0,C 180,E1 -19097.982,E2 -19097.982} C_VEL
LIN {X 0,Y 250.432,Z 416.934,A -85,B 0,C 180,E1 -19102.186,E2 -19102.186} C_VEL
LIN {X 0,Y 250.536,Z 417.31,A -85,B 0,C 180,E1 -19106.165,E2 -19106.165} C_VEL
LIN {X 0,Y 250.601,Z 418.175,A -85,B 0,C 180,E1 -19110.32,E2 -19110.32} C_VEL
LIN {X 0,Y 250.62,Z 418.435,A -85,B 0,C 180,E1 -19111.181,E2 -19111.181} C_VEL
LIN {X 0,Y 250.039,Z 419.023,A -85,B 0,C 180,E1 -19112.518,E2 -19112.518} C_VEL
LIN {X 0,Y 247.355,Z 420.497,A -85,B 0,C 180,E1 -19114.691,E2 -19114.691} C_VEL
LIN {X 0,Y 245.101,Z 421.798,A -85,B 0,C 180,E1 -19116.458,E2 -19116.458} C_VEL
LIN {X 0,Y 244.216,Z 422.656,A -85,B 0,C 180,E1 -19117.827,E2 -19117.827} C_VEL
LIN {X 0,Y 244.189,Z 422.894,A -85,B 0,C 180,E1 -19118.291,E2 -19118.291} C_VEL
LIN {X 0,Y 244.586,Z 424.719,A -85,B 0,C 180,E1 -19121.672,E2 -19121.672} C_VEL
LIN {X 0,Y 245.031,Z 427.431,A -85,B 0,C 180,E1 -19125.813,E2 -19125.813} C_VEL
LIN {X 0,Y 245.357,Z 429.922,A -85,B 0,C 180,E1 -19128.993,E2 -19128.993} C_VEL
LIN {X 0,Y 246.467,Z 433.145,A -85,B 0,C 180,E1 -19129.768,E2 -19129.768} C_VEL
LIN {X 0,Y 248.808,Z 436.739,A -85,B 0,C 180,E1 -19131.052,E2 -19131.052} C_VEL
LIN {X 0,Y 250.075,Z 440.252,A -85,B 0,C 180,E1 -19131.899,E2 -19131.899} C_VEL
LIN {X 0,Y 251.047,Z 441.961,A -85,B 0,C 180,E1 -19132.415,E2 -19132.415} C_VEL
LIN {X 0,Y 253.733,Z 451.35,A -85,B 0,C 180,E1 -19134.441,E2 -19134.441} C_VEL
LIN {X 0,Y 255.929,Z 461.245,A -85,B 0,C 180,E1 -19136.436,E2 -19136.436} C_VEL
LIN {X 0,Y 257.221,Z 471.245,A -85,B 0,C 180,E1 -19138.38,E2 -19138.38} C_VEL
LIN {X 0,Y 257.563,Z 480.867,A -85,B 0,C 180,E1 -19140.226,E2 -19140.226} C_VEL
LIN {X 0,Y 256.866,Z 491.271,A -85,B 0,C 180,E1 -19142.289,E2 -19142.289} C_VEL
LIN {X 0,Y 255.479,Z 498.946,A -85,B 0,C 180,E1 -19143.894,E2 -19143.894} C_VEL
LIN {X 0,Y 252.415,Z 507.454,A -85,B 0,C 180,E1 -19145.759,E2 -19145.759} C_VEL
LIN {X 0,Y 249.096,Z 515.972,A -85,B 0,C 180,E1 -19148.055,E2 -19148.055} C_VEL
LIN {X 0,Y 246.197,Z 523.411,A -85,B 0,C 180,E1 -19150.597,E2 -19150.597} C_VEL
LIN {X 0,Y 244.029,Z 529.531,A -85,B 0,C 180,E1 -19153.269,E2 -19153.269} C_VEL
LIN {X 0,Y 242.215,Z 533.978,A -85,B 0,C 180,E1 -19155.728,E2 -19155.728} C_VEL
LIN {X 0,Y 241.041,Z 537.422,A -85,B 0,C 180,E1 -19158.23,E2 -19158.23} C_VEL
LIN {X 0,Y 240.17,Z 540.601,A -85,B 0,C 180,E1 -19161.593,E2 -19161.593} C_VEL
LIN {X 0,Y 239.981,Z 541.59,A -85,B 0,C 180,E1 -19163.279,E2 -19163.279} C_VEL
LIN {X 0,Y 240.014,Z 542.348,A -85,B 0,C 180,E1 -19166.649,E2 -19166.649} C_VEL
LIN {X 0,Y 240.063,Z 542.141,A -85,B 0,C 180,E1 -19168.329,E2 -19168.329} C_VEL
LIN {X 0,Y 240.219,Z 541.54,A -85,B 0,C 180,E1 -19170.006,E2 -19170.006} C_VEL
LIN {X 0,Y 240.122,Z 540.452,A -85,B 0,C 180,E1 -19171.683,E2 -19171.683} C_VEL
LIN {X 0,Y 240.13,Z 538.939,A -85,B 0,C 180,E1 -19173.362,E2 -19173.362} C_VEL
LIN {X 0,Y 240.167,Z 535.996,A -85,B 0,C 180,E1 -19175.755,E2 -19175.755} C_VEL
LIN {X 0,Y 240.332,Z 531.55,A -85,B 0,C 180,E1 -19178.414,E2 -19178.414} C_VEL
LIN {X 0,Y 240.762,Z 526.067,A -85,B 0,C 180,E1 -19180.943,E2 -19180.943} C_VEL
LIN {X 0,Y 241.586,Z 519.202,A -85,B 0,C 180,E1 -19183.464,E2 -19183.464} C_VEL
LIN {X 0,Y 242.807,Z 510.607,A -85,B 0,C 180,E1 -19185.966,E2 -19185.966} C_VEL
LIN {X 0,Y 243.805,Z 503.148,A -85,B 0,C 180,E1 -19187.756,E2 -19187.756} C_VEL
LIN {X 0,Y 245.404,Z 493.456,A -85,B 0,C 180,E1 -19189.67,E2 -19189.67} C_VEL
LIN {X 0,Y 246.269,Z 487.423,A -85,B 0,C 180,E1 -19190.686,E2 -19190.686} C_VEL
LIN {X 0,Y 245.632,Z 475.932,A -85,B 0,C 180,E1 -19192.397,E2 -19192.397} C_VEL
LIN {X 0,Y 244.52,Z 463.073,A -85,B 0,C 180,E1 -19193.95,E2 -19193.95} C_VEL
LIN {X 0,Y 243.101,Z 449.597,A -85,B 0,C 180,E1 -19195.224,E2 -19195.224} C_VEL
LIN {X 0,Y 241.565,Z 437.201,A -85,B 0,C 180,E1 -19196.125,E2 -19196.125} C_VEL
LIN {X 0,Y 242.566,Z 431.691,A -85,B 0,C 180,E1 -19200.473,E2 -19200.473} C_VEL
LIN {X 0,Y 243.845,Z 425.771,A -85,B 0,C 180,E1 -19205.206,E2 -19205.206} C_VEL
LIN {X 0,Y 244.214,Z 423.348,A -85,B 0,C 180,E1 -19207.187,E2 -19207.187} C_VEL
LIN {X 0,Y 243.78,Z 419.69,A -85,B 0,C 180,E1 -19210.342,E2 -19210.342} C_VEL
LIN {X 0,Y 242.997,Z 415.675,A -85,B 0,C 180,E1 -19213.965,E2 -19213.965} C_VEL
LIN {X 0,Y 242.195,Z 411.283,A -85,B 0,C 180,E1 -19218.131,E2 -19218.131} C_VEL
LIN {X 0,Y 241.994,Z 410.345,A -85,B 0,C 180,E1 -19219.179,E2 -19219.179} C_VEL
LIN {X 0,Y 241.996,Z 410.339,A -85,B 0,C 180,E1 -19222.418,E2 -19222.418} C_VEL
LIN {X 0,Y 241.998,Z 410.338,A -85,B 0,C 180,E1 -19226.509,E2 -19226.509} C_VEL
LIN {X 0,Y 241.996,Z 410.34,A -85,B 0,C 180,E1 -19230.614,E2 -19230.614} C_VEL
LIN {X 0,Y 242.052,Z 410.33,A -85,B 0,C 180,E1 -19234.18,E2 -19234.18} C_VEL
LIN {X 0,Y 242.011,Z 410.337,A -85,B 0,C 180,E1 -19238.335,E2 -19238.335} C_VEL
LIN {X 0,Y 242.133,Z 410.323,A -85,B 0,C 180,E1 -19243.318,E2 -19243.318} C_VEL
LIN {X 0,Y 242.183,Z 410.315,A -85,B 0,C 180,E1 -19248.278,E2 -19248.278} C_VEL
LIN {X 0,Y 242.404,Z 410.287,A -85,B 0,C 180,E1 -19251.663,E2 -19251.663} C_VEL
LIN {X 0,Y 242.26,Z 410.309,A -85,B 0,C 180,E1 -19255.006,E2 -19255.006} C_VEL
LIN {X 0,Y 242.649,Z 410.256,A -85,B 0,C 180,E1 -19258.339,E2 -19258.339} C_VEL
LIN {X 0,Y 242.639,Z 410.259,A -85,B 0,C 180,E1 -19261.658,E2 -19261.658} C_VEL
LIN {X 0,Y 242.413,Z 410.288,A -85,B 0,C 180,E1 -19266.658,E2 -19266.658} C_VEL
LIN {X 0,Y 242.278,Z 410.303,A -85,B 0,C 180,E1 -19270.022,E2 -19270.022} C_VEL
LIN {X 0,Y 242.136,Z 410.321,A -85,B 0,C 180,E1 -19275.141,E2 -19275.141} C_VEL
LIN {X 0,Y 242.046,Z 410.336,A -85,B 0,C 180,E1 -19278.625,E2 -19278.625} C_VEL
LIN {X 0,Y 242.003,Z 410.338,A -85,B 0,C 180,E1 -19282.179,E2 -19282.179} C_VEL
LIN {X 0,Y 242.081,Z 410.328,A -85,B 0,C 180,E1 -19285.835,E2 -19285.835} C_VEL
LIN {X 0,Y 241.989,Z 410.339,A -85,B 0,C 180,E1 -19289.584,E2 -19289.584} C_VEL
LIN {X 0,Y 241.991,Z 410.338,A -85,B 0,C 180,E1 -19293.489,E2 -19293.489} C_VEL
LIN {X 0,Y 241.999,Z 410.338,A -85,B 0,C 180,E1 -19297.578,E2 -19297.578} C_VEL
LIN {X 0,Y 241.943,Z 410.345,A -85,B 0,C 180,E1 -19301.919,E2 -19301.919} C_VEL
LIN {X 0,Y 241.932,Z 410.349,A -85,B 0,C 180,E1 -19306.569,E2 -19306.569} C_VEL
LIN {X 0,Y 242.002,Z 410.338,A -85,B 0,C 180,E1 -19311.635,E2 -19311.635} C_VEL
LIN {X 0,Y 241.988,Z 410.343,A -85,B 0,C 180,E1 -19314.483,E2 -19314.483} C_VEL
LIN {X 0,Y 241.98,Z 410.344,A -85,B 0,C 180,E1 -19318.475,E2 -19318.475} C_VEL
LIN {X 0,Y 242.011,Z 410.341,A -85,B 0,C 180,E1 -19322.307,E2 -19322.307} C_VEL
LIN {X 0,Y 242.061,Z 410.33,A -85,B 0,C 180,E1 -19326.011,E2 -19326.011} C_VEL
LIN {X 0,Y 242.04,Z 410.334,A -85,B 0,C 180,E1 -19329.602,E2 -19329.602} C_VEL
LIN {X 0,Y 242.164,Z 410.315,A -85,B 0,C 180,E1 -19333.272,E2 -19333.272} C_VEL
LIN {X 0,Y 242.179,Z 410.32,A -85,B 0,C 180,E1 -19338.274,E2 -19338.274} C_VEL
LIN {X 0,Y 242.397,Z 410.288,A -85,B 0,C 180,E1 -19341.659,E2 -19341.659} C_VEL
LIN {X 0,Y 242.251,Z 410.307,A -85,B 0,C 180,E1 -19345.001,E2 -19345.001} C_VEL
LIN {X 0,Y 242.629,Z 410.262,A -85,B 0,C 180,E1 -19348.334,E2 -19348.334} C_VEL
LIN {X 0,Y 242.629,Z 410.259,A -85,B 0,C 180,E1 -19351.654,E2 -19351.654} C_VEL
LIN {X 0,Y 242.424,Z 410.285,A -85,B 0,C 180,E1 -19356.653,E2 -19356.653} C_VEL
LIN {X 0,Y 242.334,Z 410.298,A -85,B 0,C 180,E1 -19360.014,E2 -19360.014} C_VEL
LIN {X 0,Y 242.154,Z 410.318,A -85,B 0,C 180,E1 -19365.135,E2 -19365.135} C_VEL
LIN {X 0,Y 242.058,Z 410.331,A -85,B 0,C 180,E1 -19368.618,E2 -19368.618} C_VEL
LIN {X 0,Y 241.975,Z 410.344,A -85,B 0,C 180,E1 -19372.176,E2 -19372.176} C_VEL
LIN {X 0,Y 241.881,Z 410.356,A -85,B 0,C 180,E1 -19375.831,E2 -19375.831} C_VEL
LIN {X 0,Y 241.52,Z 410.401,A -85,B 0,C 180,E1 -19379.641,E2 -19379.641} C_VEL
LIN {X 0,Y 240.992,Z 410.467,A -85,B 0,C 180,E1 -19383.64,E2 -19383.64} C_VEL
LIN {X 0,Y 240.793,Z 410.721,A -85,B 0,C 180,E1 -19385.705,E2 -19385.705} C_VEL
LIN {X 0,Y 240.772,Z 410.939,A -85,B 0,C 180,E1 -19385.999,E2 -19385.999} C_VEL
LIN {X 0,Y 244.07,Z 424.799,A -85,B 0,C 180,E1 -19387.198,E2 -19387.198} C_VEL
LIN {X 0,Y 246.829,Z 437.481,A -85,B 0,C 180,E1 -19388.58,E2 -19388.58} C_VEL
LIN {X 0,Y 248.787,Z 448.314,A -85,B 0,C 180,E1 -19390.001,E2 -19390.001} C_VEL
LIN {X 0,Y 247.457,Z 458.912,A -85,B 0,C 180,E1 -19391.492,E2 -19391.492} C_VEL
LIN {X 0,Y 245.812,Z 470.255,A -85,B 0,C 180,E1 -19393.475,E2 -19393.475} C_VEL
LIN {X 0,Y 244.448,Z 479.47,A -85,B 0,C 180,E1 -19395.464,E2 -19395.464} C_VEL
LIN {X 0,Y 243.036,Z 488.106,A -85,B 0,C 180,E1 -19397.755,E2 -19397.755} C_VEL
LIN {X 0,Y 241.96,Z 495.8,A -85,B 0,C 180,E1 -19400.284,E2 -19400.284} C_VEL
LIN {X 0,Y 241.092,Z 501.909,A -85,B 0,C 180,E1 -19402.782,E2 -19402.782} C_VEL
LIN {X 0,Y 240.51,Z 507.215,A -85,B 0,C 180,E1 -19405.557,E2 -19405.557} C_VEL
LIN {X 0,Y 240.069,Z 511,A -85,B 0,C 180,E1 -19408.203,E2 -19408.203} C_VEL
LIN {X 0,Y 239.838,Z 514.187,A -85,B 0,C 180,E1 -19411.517,E2 -19411.517} C_VEL
LIN {X 0,Y 240.141,Z 515.866,A -85,B 0,C 180,E1 -19415.109,E2 -19415.109} C_VEL
LIN {X 0,Y 240.671,Z 515.958,A -85,B 0,C 180,E1 -19417.692,E2 -19417.692} C_VEL
LIN {X 0,Y 241.306,Z 515.426,A -85,B 0,C 180,E1 -19419.545,E2 -19419.545} C_VEL
LIN {X 0,Y 242.725,Z 513.346,A -85,B 0,C 180,E1 -19422.817,E2 -19422.817} C_VEL
LIN {X 0,Y 244.631,Z 509.891,A -85,B 0,C 180,E1 -19425.867,E2 -19425.867} C_VEL
LIN {X 0,Y 246.751,Z 505.632,A -85,B 0,C 180,E1 -19428.501,E2 -19428.501} C_VEL
LIN {X 0,Y 249.106,Z 500.604,A -85,B 0,C 180,E1 -19430.864,E2 -19430.864} C_VEL
LIN {X 0,Y 251.835,Z 494.395,A -85,B 0,C 180,E1 -19433.19,E2 -19433.19} C_VEL
LIN {X 0,Y 255.213,Z 486.021,A -85,B 0,C 180,E1 -19435.658,E2 -19435.658} C_VEL
LIN {X 0,Y 258.44,Z 477.348,A -85,B 0,C 180,E1 -19437.664,E2 -19437.664} C_VEL
LIN {X 0,Y 261.866,Z 466.86,A -85,B 0,C 180,E1 -19439.617,E2 -19439.617} C_VEL
LIN {X 0,Y 261.755,Z 461.932,A -85,B 0,C 180,E1 -19440.736,E2 -19440.736} C_VEL
LIN {X 0,Y 259.522,Z 451.002,A -85,B 0,C 180,E1 -19443.391,E2 -19443.391} C_VEL
LIN {X 0,Y 257.581,Z 444.03,A -85,B 0,C 180,E1 -19445.132,E2 -19445.132} C_VEL
LIN {X 0,Y 254.515,Z 436.853,A -85,B 0,C 180,E1 -19447.139,E2 -19447.139} C_VEL
LIN {X 0,Y 251.639,Z 431.571,A -85,B 0,C 180,E1 -19448.837,E2 -19448.837} C_VEL
LIN {X 0,Y 250.276,Z 428.784,A -85,B 0,C 180,E1 -19449.701,E2 -19449.701} C_VEL
LIN {X 0,Y 247.829,Z 425.432,A -85,B 0,C 180,E1 -19451.088,E2 -19451.088} C_VEL
LIN {X 0,Y 247.011,Z 423.958,A -85,B 0,C 180,E1 -19451.594,E2 -19451.594} C_VEL
LIN {X 0,Y 244.635,Z 421.554,A -85,B 0,C 180,E1 -19452.919,E2 -19452.919} C_VEL
LIN {X 0,Y 243.576,Z 419.008,A -85,B 0,C 180,E1 -19453.772,E2 -19453.772} C_VEL
LIN {X 0,Y 243.539,Z 418.587,A -85,B 0,C 180,E1 -19457.793,E2 -19457.793} C_VEL
LIN {X 0,Y 243.543,Z 418.575,A -85,B 0,C 180,E1 -19462.035,E2 -19462.035} C_VEL
LIN {X 0,Y 243.614,Z 419.04,A -85,B 0,C 180,E1 -19466.596,E2 -19466.596} C_VEL
LIN {X 0,Y 243.696,Z 419.786,A -85,B 0,C 180,E1 -19470.113,E2 -19470.113} C_VEL
LIN {X 0,Y 243.852,Z 420.769,A -85,B 0,C 180,E1 -19473.314,E2 -19473.314} C_VEL
LIN {X 0,Y 244.102,Z 422.374,A -85,B 0,C 180,E1 -19477.203,E2 -19477.203} C_VEL
LIN {X 0,Y 244.189,Z 422.894,A -85,B 0,C 180,E1 -19478.291,E2 -19478.291} C_VEL
LIN {X 0,Y 243.642,Z 423.502,A -85,B 0,C 180,E1 -19479.2,E2 -19479.2} C_VEL
LIN {X 0,Y 241.038,Z 424.911,A -85,B 0,C 180,E1 -19480.624,E2 -19480.624} C_VEL
LIN {X 0,Y 238.372,Z 426.381,A -85,B 0,C 180,E1 -19482.076,E2 -19482.076} C_VEL
LIN {X 0,Y 237.77,Z 427.097,A -85,B 0,C 180,E1 -19483.015,E2 -19483.015} C_VEL
LIN {X 0,Y 238.069,Z 428.82,A -85,B 0,C 180,E1 -19485.49,E2 -19485.49} C_VEL
LIN {X 0,Y 239.656,Z 432.77,A -85,B 0,C 180,E1 -19486.83,E2 -19486.83} C_VEL
LIN {X 0,Y 242.067,Z 436.04,A -85,B 0,C 180,E1 -19488.385,E2 -19488.385} C_VEL
LIN {X 0,Y 243.299,Z 439.347,A -85,B 0,C 180,E1 -19489.349,E2 -19489.349} C_VEL
LIN {X 0,Y 244.725,Z 441.515,A -85,B 0,C 180,E1 -19490.195,E2 -19490.195} C_VEL
LIN {X 0,Y 246.079,Z 445.329,A -85,B 0,C 180,E1 -19491.231,E2 -19491.231} C_VEL
LIN {X 0,Y 246.861,Z 446.97,A -85,B 0,C 180,E1 -19491.751,E2 -19491.751} C_VEL
LIN {X 0,Y 248.964,Z 455.288,A -85,B 0,C 180,E1 -19493.652,E2 -19493.652} C_VEL
LIN {X 0,Y 251.008,Z 467.431,A -85,B 0,C 180,E1 -19496.265,E2 -19496.265} C_VEL
LIN {X 0,Y 251.68,Z 477.588,A -85,B 0,C 180,E1 -19498.371,E2 -19498.371} C_VEL
LIN {X 0,Y 251.321,Z 487.906,A -85,B 0,C 180,E1 -19500.505,E2 -19500.505} C_VEL
LIN {X 0,Y 250.04,Z 496.561,A -85,B 0,C 180,E1 -19502.377,E2 -19502.377} C_VEL
LIN {X 0,Y 249.217,Z 500.137,A -85,B 0,C 180,E1 -19503.187,E2 -19503.187} C_VEL
LIN {X 0,Y 245.452,Z 509.83,A -85,B 0,C 180,E1 -19505.477,E2 -19505.477} C_VEL
LIN {X 0,Y 242.032,Z 517.828,A -85,B 0,C 180,E1 -19507.829,E2 -19507.829} C_VEL
LIN {X 0,Y 238.946,Z 525.24,A -85,B 0,C 180,E1 -19510.629,E2 -19510.629} C_VEL
LIN {X 0,Y 237.233,Z 529.734,A -85,B 0,C 180,E1 -19512.775,E2 -19512.775} C_VEL
LIN {X 0,Y 235.326,Z 534.038,A -85,B 0,C 180,E1 -19515.301,E2 -19515.301} C_VEL
LIN {X 0,Y 234.065,Z 537.342,A -85,B 0,C 180,E1 -19517.874,E2 -19517.874} C_VEL
LIN {X 0,Y 233.496,Z 539.052,A -85,B 0,C 180,E1 -19519.602,E2 -19519.602} C_VEL
LIN {X 0,Y 233.113,Z 540.353,A -85,B 0,C 180,E1 -19521.337,E2 -19521.337} C_VEL
LIN {X 0,Y 232.842,Z 541.76,A -85,B 0,C 180,E1 -19524.811,E2 -19524.811} C_VEL
LIN {X 0,Y 232.923,Z 541.892,A -85,B 0,C 180,E1 -19526.547,E2 -19526.547} C_VEL
LIN {X 0,Y 232.989,Z 541.626,A -85,B 0,C 180,E1 -19528.278,E2 -19528.278} C_VEL
LIN {X 0,Y 233.141,Z 540.92,A -85,B 0,C 180,E1 -19530.006,E2 -19530.006} C_VEL
LIN {X 0,Y 233.048,Z 539.771,A -85,B 0,C 180,E1 -19531.734,E2 -19531.734} C_VEL
LIN {X 0,Y 233.067,Z 537.241,A -85,B 0,C 180,E1 -19534.33,E2 -19534.33} C_VEL
LIN {X 0,Y 233.132,Z 533.635,A -85,B 0,C 180,E1 -19536.932,E2 -19536.932} C_VEL
LIN {X 0,Y 233.407,Z 528.86,A -85,B 0,C 180,E1 -19539.539,E2 -19539.539} C_VEL
LIN {X 0,Y 233.974,Z 522.776,A -85,B 0,C 180,E1 -19542.144,E2 -19542.144} C_VEL
LIN {X 0,Y 235.084,Z 515.228,A -85,B 0,C 180,E1 -19544.727,E2 -19544.727} C_VEL
LIN {X 0,Y 236.127,Z 507.476,A -85,B 0,C 180,E1 -19546.876,E2 -19546.876} C_VEL
LIN {X 0,Y 237.643,Z 498.116,A -85,B 0,C 180,E1 -19548.99,E2 -19548.99} C_VEL
LIN {X 0,Y 239.227,Z 487.863,A -85,B 0,C 180,E1 -19550.873,E2 -19550.873} C_VEL
LIN {X 0,Y 238.643,Z 476.437,A -85,B 0,C 180,E1 -19552.663,E2 -19552.663} C_VEL
LIN {X 0,Y 237.542,Z 463.059,A -85,B 0,C 180,E1 -19554.345,E2 -19554.345} C_VEL
LIN {X 0,Y 236.11,Z 449.641,A -85,B 0,C 180,E1 -19555.674,E2 -19555.674} C_VEL
LIN {X 0,Y 234.58,Z 436.848,A -85,B 0,C 180,E1 -19556.62,E2 -19556.62} C_VEL
LIN {X 0,Y 235.671,Z 430.923,A -85,B 0,C 180,E1 -19561.464,E2 -19561.464} C_VEL
LIN {X 0,Y 236.802,Z 426.204,A -85,B 0,C 180,E1 -19565.368,E2 -19565.368} C_VEL
LIN {X 0,Y 237.113,Z 424.456,A -85,B 0,C 180,E1 -19566.842,E2 -19566.842} C_VEL
LIN {X 0,Y 236.887,Z 421.41,A -85,B 0,C 180,E1 -19569.521,E2 -19569.521} C_VEL
LIN {X 0,Y 236.126,Z 417.395,A -85,B 0,C 180,E1 -19573.208,E2 -19573.208} C_VEL
LIN {X 0,Y 235.43,Z 413.835,A -85,B 0,C 180,E1 -19576.637,E2 -19576.637} C_VEL
LIN {X 0,Y 234.943,Z 411.22,A -85,B 0,C 180,E1 -19579.41,E2 -19579.41} C_VEL
LIN {X 0,Y 234.938,Z 411.216,A -85,B 0,C 180,E1 -19583.879,E2 -19583.879} C_VEL
LIN {X 0,Y 234.972,Z 411.216,A -85,B 0,C 180,E1 -19587.425,E2 -19587.425} C_VEL
LIN {X 0,Y 234.921,Z 411.221,A -85,B 0,C 180,E1 -19591.4,E2 -19591.4} C_VEL
LIN {X 0,Y 234.972,Z 411.217,A -85,B 0,C 180,E1 -19595.243,E2 -19595.243} C_VEL
LIN {X 0,Y 234.962,Z 411.219,A -85,B 0,C 180,E1 -19598.964,E2 -19598.964} C_VEL
LIN {X 0,Y 235.074,Z 411.203,A -85,B 0,C 180,E1 -19603.093,E2 -19603.093} C_VEL
LIN {X 0,Y 235.115,Z 411.195,A -85,B 0,C 180,E1 -19607.921,E2 -19607.921} C_VEL
LIN {X 0,Y 235.337,Z 411.169,A -85,B 0,C 180,E1 -19611.411,E2 -19611.411} C_VEL
LIN {X 0,Y 235.377,Z 411.166,A -85,B 0,C 180,E1 -19613.139,E2 -19613.139} C_VEL
LIN {X 0,Y 235.609,Z 411.133,A -85,B 0,C 180,E1 -19618.289,E2 -19618.289} C_VEL
LIN {X 0,Y 235.597,Z 411.136,A -85,B 0,C 180,E1 -19621.708,E2 -19621.708} C_VEL
LIN {X 0,Y 235.364,Z 411.166,A -85,B 0,C 180,E1 -19626.858,E2 -19626.858} C_VEL
LIN {X 0,Y 235.226,Z 411.183,A -85,B 0,C 180,E1 -19630.325,E2 -19630.325} C_VEL
LIN {X 0,Y 235.085,Z 411.197,A -85,B 0,C 180,E1 -19635.607,E2 -19635.607} C_VEL
LIN {X 0,Y 234.985,Z 411.213,A -85,B 0,C 180,E1 -19639.206,E2 -19639.206} C_VEL
LIN {X 0,Y 234.958,Z 411.216,A -85,B 0,C 180,E1 -19642.881,E2 -19642.881} C_VEL
LIN {X 0,Y 234.978,Z 411.216,A -85,B 0,C 180,E1 -19646.654,E2 -19646.654} C_VEL
LIN {X 0,Y 234.915,Z 411.223,A -85,B 0,C 180,E1 -19650.568,E2 -19650.568} C_VEL
LIN {X 0,Y 234.941,Z 411.221,A -85,B 0,C 180,E1 -19654.634,E2 -19654.634} C_VEL
LIN {X 0,Y 234.953,Z 411.216,A -85,B 0,C 180,E1 -19658.94,E2 -19658.94} C_VEL
LIN {X 0,Y 234.888,Z 411.224,A -85,B 0,C 180,E1 -19663.483,E2 -19663.483} C_VEL
LIN {X 0,Y 234.885,Z 411.227,A -85,B 0,C 180,E1 -19666.507,E2 -19666.507} C_VEL
LIN {X 0,Y 234.925,Z 411.22,A -85,B 0,C 180,E1 -19671.073,E2 -19671.073} C_VEL
LIN {X 0,Y 234.933,Z 411.217,A -85,B 0,C 180,E1 -19675.356,E2 -19675.356} C_VEL
LIN {X 0,Y 234.936,Z 411.218,A -85,B 0,C 180,E1 -19679.427,E2 -19679.427} C_VEL
LIN {X 0,Y 234.998,Z 411.21,A -85,B 0,C 180,E1 -19683.788,E2 -19683.788} C_VEL
LIN {X 0,Y 235.014,Z 411.209,A -85,B 0,C 180,E1 -19688.964,E2 -19688.964} C_VEL
LIN {X 0,Y 235.097,Z 411.196,A -85,B 0,C 180,E1 -19693.053,E2 -19693.053} C_VEL
LIN {X 0,Y 235.113,Z 411.198,A -85,B 0,C 180,E1 -19697.916,E2 -19697.916} C_VEL
LIN {X 0,Y 235.328,Z 411.167,A -85,B 0,C 180,E1 -19701.406,E2 -19701.406} C_VEL
LIN {X 0,Y 235.37,Z 411.163,A -85,B 0,C 180,E1 -19703.134,E2 -19703.134} C_VEL
LIN {X 0,Y 235.589,Z 411.139,A -85,B 0,C 180,E1 -19708.284,E2 -19708.284} C_VEL
LIN {X 0,Y 235.589,Z 411.136,A -85,B 0,C 180,E1 -19711.703,E2 -19711.703} C_VEL
LIN {X 0,Y 235.396,Z 411.16,A -85,B 0,C 180,E1 -19716.852,E2 -19716.852} C_VEL
LIN {X 0,Y 235.242,Z 411.182,A -85,B 0,C 180,E1 -19720.32,E2 -19720.32} C_VEL
LIN {X 0,Y 235.1,Z 411.198,A -85,B 0,C 180,E1 -19725.6,E2 -19725.6} C_VEL
LIN {X 0,Y 234.993,Z 411.21,A -85,B 0,C 180,E1 -19729.2,E2 -19729.2} C_VEL
LIN {X 0,Y 234.908,Z 411.221,A -85,B 0,C 180,E1 -19732.881,E2 -19732.881} C_VEL
LIN {X 0,Y 234.746,Z 411.242,A -85,B 0,C 180,E1 -19736.677,E2 -19736.677} C_VEL
LIN {X 0,Y 234.326,Z 411.295,A -85,B 0,C 180,E1 -19740.647,E2 -19740.647} C_VEL
LIN {X 0,Y 233.763,Z 411.374,A -85,B 0,C 180,E1 -19745.49,E2 -19745.49} C_VEL
LIN {X 0,Y 237.53,Z 427.403,A -85,B 0,C 180,E1 -19746.955,E2 -19746.955} C_VEL
LIN {X 0,Y 240.223,Z 440.077,A -85,B 0,C 180,E1 -19748.431,E2 -19748.431} C_VEL
LIN {X 0,Y 241.825,Z 449.5,A -85,B 0,C 180,E1 -19749.735,E2 -19749.735} C_VEL
LIN {X 0,Y 240.287,Z 460.687,A -85,B 0,C 180,E1 -19751.385,E2 -19751.385} C_VEL
LIN {X 0,Y 238.782,Z 470.894,A -85,B 0,C 180,E1 -19753.245,E2 -19753.245} C_VEL
LIN {X 0,Y 237.397,Z 479.944,A -85,B 0,C 180,E1 -19755.265,E2 -19755.265} C_VEL
LIN {X 0,Y 235.993,Z 488.412,A -85,B 0,C 180,E1 -19757.583,E2 -19757.583} C_VEL
LIN {X 0,Y 234.948,Z 495.549,A -85,B 0,C 180,E1 -19759.977,E2 -19759.977} C_VEL
LIN {X 0,Y 234.039,Z 501.857,A -85,B 0,C 180,E1 -19762.592,E2 -19762.592} C_VEL
LIN {X 0,Y 233.48,Z 506.701,A -85,B 0,C 180,E1 -19765.118,E2 -19765.118} C_VEL
LIN {X 0,Y 233.092,Z 510.387,A -85,B 0,C 180,E1 -19767.575,E2 -19767.575} C_VEL
LIN {X 0,Y 232.881,Z 512.253,A -85,B 0,C 180,E1 -19769.136,E2 -19769.136} C_VEL
LIN {X 0,Y 232.743,Z 514.119,A -85,B 0,C 180,E1 -19771.111,E2 -19771.111} C_VEL
LIN {X 0,Y 232.813,Z 515.41,A -85,B 0,C 180,E1 -19773.078,E2 -19773.078} C_VEL
LIN {X 0,Y 233.042,Z 516.221,A -85,B 0,C 180,E1 -19775.028,E2 -19775.028} C_VEL
LIN {X 0,Y 233.394,Z 516.483,A -85,B 0,C 180,E1 -19776.957,E2 -19776.957} C_VEL
LIN {X 0,Y 233.949,Z 516.284,A -85,B 0,C 180,E1 -19778.872,E2 -19778.872} C_VEL
LIN {X 0,Y 234.67,Z 515.624,A -85,B 0,C 180,E1 -19780.767,E2 -19780.767} C_VEL
LIN {X 0,Y 235.561,Z 514.438,A -85,B 0,C 180,E1 -19782.666,E2 -19782.666} C_VEL
LIN {X 0,Y 237.201,Z 511.846,A -85,B 0,C 180,E1 -19785.415,E2 -19785.415} C_VEL
LIN {X 0,Y 239.285,Z 508.12,A -85,B 0,C 180,E1 -19788.137,E2 -19788.137} C_VEL
LIN {X 0,Y 241.964,Z 503.008,A -85,B 0,C 180,E1 -19790.899,E2 -19790.899} C_VEL
LIN {X 0,Y 244.867,Z 496.938,A -85,B 0,C 180,E1 -19793.409,E2 -19793.409} C_VEL
LIN {X 0,Y 248.407,Z 488.977,A -85,B 0,C 180,E1 -19795.946,E2 -19795.946} C_VEL
LIN {X 0,Y 251.687,Z 480.922,A -85,B 0,C 180,E1 -19798.001,E2 -19798.001} C_VEL
LIN {X 0,Y 255.275,Z 471.167,A -85,B 0,C 180,E1 -19800.001,E2 -19800.001} C_VEL
LIN {X 0,Y 256.048,Z 468.643,A -85,B 0,C 180,E1 -19800.459,E2 -19800.459} C_VEL
LIN {X 0,Y 255.712,Z 463.059,A -85,B 0,C 180,E1 -19801.863,E2 -19801.863} C_VEL
LIN {X 0,Y 253.625,Z 451.878,A -85,B 0,C 180,E1 -19804.77,E2 -19804.77} C_VEL
LIN {X 0,Y 251.757,Z 446.073,A -85,B 0,C 180,E1 -19806.413,E2 -19806.413} C_VEL
LIN {X 0,Y 248.287,Z 437.993,A -85,B 0,C 180,E1 -19808.958,E2 -19808.958} C_VEL
LIN {X 0,Y 245.481,Z 433.138,A -85,B 0,C 180,E1 -19810.829,E2 -19810.829} C_VEL
LIN {X 0,Y 244.077,Z 430.643,A -85,B 0,C 180,E1 -19811.8,E2 -19811.8} C_VEL
LIN {X 0,Y 241.518,Z 427.478,A -85,B 0,C 180,E1 -19813.463,E2 -19813.463} C_VEL
